//     RulliCentroTagliTask Inputs/RULLI_CENTRO_TAGLI.Catenaria_C4_Rotazione_Status_Dword/InTargetPosition <-> Outputs/ToPlc/StateDWord/InTargetPosition
//     RulliCentroTagliTask Inputs/RULLI_CENTRO_TAGLI.Catenaria_C4_Rotazione_Status_Dword/IoDataInvalid <-> Outputs/ToPlc/StateDWord/IoDataInvalid
//     RulliCentroTagliTask Inputs/RULLI_CENTRO_TAGLI.Catenaria_C4_Rotazione_Status_Dword/MotionCommandsLocked <-> Outputs/ToPlc/StateDWord/MotionCommandsLocked
//     RulliCentroTagliTask Inputs/RULLI_CENTRO_TAGLI.Catenaria_C4_Rotazione_Status_Dword/NegativeDirection <-> Outputs/ToPlc/StateDWord/NegativeDirection
//     RulliCentroTagliTask Inputs/RULLI_CENTRO_TAGLI.Catenaria_C4_Rotazione_Status_Dword/NewTargetPos <-> Outputs/ToPlc/StateDWord/NewTargetPos
//     RulliCentroTagliTask Inputs/RULLI_CENTRO_TAGLI.Catenaria_C4_Rotazione_Status_Dword/NotMoving <-> Outputs/ToPlc/StateDWord/NotMoving
//     RulliCentroTagliTask Inputs/RULLI_CENTRO_TAGLI.Catenaria_C4_Rotazione_Status_Dword/Operational <-> Outputs/ToPlc/StateDWord/Operational
//     RulliCentroTagliTask Inputs/RULLI_CENTRO_TAGLI.Catenaria_C4_Rotazione_Status_Dword/PTPmode <-> Outputs/ToPlc/StateDWord/PTPmode
//     RulliCentroTagliTask Inputs/RULLI_CENTRO_TAGLI.Catenaria_C4_Rotazione_Status_Dword/PhasingActive <-> Outputs/ToPlc/StateDWord/PhasingActive
//     RulliCentroTagliTask Inputs/RULLI_CENTRO_TAGLI.Catenaria_C4_Rotazione_Status_Dword/PositiveDirection <-> Outputs/ToPlc/StateDWord/PositiveDirection
//     RulliCentroTagliTask Inputs/RULLI_CENTRO_TAGLI.Catenaria_C4_Rotazione_Status_Dword/Protected_ <-> Outputs/ToPlc/StateDWord/Protected
//     RulliCentroTagliTask Inputs/RULLI_CENTRO_TAGLI.Catenaria_C4_Rotazione_Status_Dword/SoftLimitMaxExceeded <-> Outputs/ToPlc/StateDWord/SoftLimitMaxExceeded
//     RulliCentroTagliTask Inputs/RULLI_CENTRO_TAGLI.Catenaria_C4_Rotazione_Status_Dword/SoftLimitMinExceeded <-> Outputs/ToPlc/StateDWord/SoftLimitMinExceeded
//     RulliCentroTagliTask Outputs/RULLI_CENTRO_TAGLI.Catenaria_C4_Rotazione.PlcToNc <-> Inputs/FromPlc
//   Galimberti/Galimberti Instance <-> NC-Task 1 SAF/Axes/C5
//     RulliCentroTagliTask Inputs/RULLI_CENTRO_TAGLI.Catenaria_C5_Rotazione.NcToPlc <-> Outputs/ToPlc
//     RulliCentroTagliTask Inputs/RULLI_CENTRO_TAGLI.Catenaria_C5_Rotazione_Status_Dword/CamDataQueued <-> Outputs/ToPlc/StateDWord/CamDataQueued
//     RulliCentroTagliTask Inputs/RULLI_CENTRO_TAGLI.Catenaria_C5_Rotazione_Status_Dword/CamScalingPending <-> Outputs/ToPlc/StateDWord/CamScalingPending
//     RulliCentroTagliTask Inputs/RULLI_CENTRO_TAGLI.Catenaria_C5_Rotazione_Status_Dword/CamTableQueued <-> Outputs/ToPlc/StateDWord/CamTableQueued
//     RulliCentroTagliTask Inputs/RULLI_CENTRO_TAGLI.Catenaria_C5_Rotazione_Status_Dword/CmdBuffered <-> Outputs/ToPlc/StateDWord/CmdBuffered
//     RulliCentroTagliTask Inputs/RULLI_CENTRO_TAGLI.Catenaria_C5_Rotazione_Status_Dword/Compensating <-> Outputs/ToPlc/StateDWord/Compensating
//     RulliCentroTagliTask Inputs/RULLI_CENTRO_TAGLI.Catenaria_C5_Rotazione_Status_Dword/ConstantVelocity <-> Outputs/ToPlc/StateDWord/ConstantVelocity
//     RulliCentroTagliTask Inputs/RULLI_CENTRO_TAGLI.Catenaria_C5_Rotazione_Status_Dword/ContinuousMotion <-> Outputs/ToPlc/StateDWord/ContinuousMotion
//     RulliCentroTagliTask Inputs/RULLI_CENTRO_TAGLI.Catenaria_C5_Rotazione_Status_Dword/ControlLoopClosed <-> Outputs/ToPlc/StateDWord/ControlLoopClosed
//     RulliCentroTagliTask Inputs/RULLI_CENTRO_TAGLI.Catenaria_C5_Rotazione_Status_Dword/DriveDeviceError <-> Outputs/ToPlc/StateDWord/DriveDeviceError
//     RulliCentroTagliTask Inputs/RULLI_CENTRO_TAGLI.Catenaria_C5_Rotazione_Status_Dword/Error <-> Outputs/ToPlc/StateDWord/Error
//     RulliCentroTagliTask Inputs/RULLI_CENTRO_TAGLI.Catenaria_C5_Rotazione_Status_Dword/ErrorPropagationDelayed <-> Outputs/ToPlc/StateDWord/ErrorPropagationDelayed
//     RulliCentroTagliTask Inputs/RULLI_CENTRO_TAGLI.Catenaria_C5_Rotazione_Status_Dword/ExtSetPointGenEnabled <-> Outputs/ToPlc/StateDWord/ExtSetPointGenEnabled
//     RulliCentroTagliTask Inputs/RULLI_CENTRO_TAGLI.Catenaria_C5_Rotazione_Status_Dword/ExternalLatchValid <-> Outputs/ToPlc/StateDWord/ExternalLatchValid
//     RulliCentroTagliTask Inputs/RULLI_CENTRO_TAGLI.Catenaria_C5_Rotazione_Status_Dword/HasBeenStopped <-> Outputs/ToPlc/StateDWord/HasBeenStopped
//     RulliCentroTagliTask Inputs/RULLI_CENTRO_TAGLI.Catenaria_C5_Rotazione_Status_Dword/HasJob <-> Outputs/ToPlc/StateDWord/HasJob
//     RulliCentroTagliTask Inputs/RULLI_CENTRO_TAGLI.Catenaria_C5_Rotazione_Status_Dword/Homed <-> Outputs/ToPlc/StateDWord/Homed
//     RulliCentroTagliTask Inputs/RULLI_CENTRO_TAGLI.Catenaria_C5_Rotazione_Status_Dword/HomingBusy <-> Outputs/ToPlc/StateDWord/HomingBusy
//     RulliCentroTagliTask Inputs/RULLI_CENTRO_TAGLI.Catenaria_C5_Rotazione_Status_Dword/InPositionArea <-> Outputs/ToPlc/StateDWord/InPositionArea
//     RulliCentroTagliTask Inputs/RULLI_CENTRO_TAGLI.Catenaria_C5_Rotazione_Status_Dword/InTargetPosition <-> Outputs/ToPlc/StateDWord/InTargetPosition
//     RulliCentroTagliTask Inputs/RULLI_CENTRO_TAGLI.Catenaria_C5_Rotazione_Status_Dword/IoDataInvalid <-> Outputs/ToPlc/StateDWord/IoDataInvalid
//     RulliCentroTagliTask Inputs/RULLI_CENTRO_TAGLI.Catenaria_C5_Rotazione_Status_Dword/MotionCommandsLocked <-> Outputs/ToPlc/StateDWord/MotionCommandsLocked
//     RulliCentroTagliTask Inputs/RULLI_CENTRO_TAGLI.Catenaria_C5_Rotazione_Status_Dword/NegativeDirection <-> Outputs/ToPlc/StateDWord/NegativeDirection
//     RulliCentroTagliTask Inputs/RULLI_CENTRO_TAGLI.Catenaria_C5_Rotazione_Status_Dword/NewTargetPos <-> Outputs/ToPlc/StateDWord/NewTargetPos
//     RulliCentroTagliTask Inputs/RULLI_CENTRO_TAGLI.Catenaria_C5_Rotazione_Status_Dword/NotMoving <-> Outputs/ToPlc/StateDWord/NotMoving
//     RulliCentroTagliTask Inputs/RULLI_CENTRO_TAGLI.Catenaria_C5_Rotazione_Status_Dword/Operational <-> Outputs/ToPlc/StateDWord/Operational
//     RulliCentroTagliTask Inputs/RULLI_CENTRO_TAGLI.Catenaria_C5_Rotazione_Status_Dword/PTPmode <-> Outputs/ToPlc/StateDWord/PTPmode
//     RulliCentroTagliTask Inputs/RULLI_CENTRO_TAGLI.Catenaria_C5_Rotazione_Status_Dword/PhasingActive <-> Outputs/ToPlc/StateDWord/PhasingActive
//     RulliCentroTagliTask Inputs/RULLI_CENTRO_TAGLI.Catenaria_C5_Rotazione_Status_Dword/PositiveDirection <-> Outputs/ToPlc/StateDWord/PositiveDirection
//     RulliCentroTagliTask Inputs/RULLI_CENTRO_TAGLI.Catenaria_C5_Rotazione_Status_Dword/Protected_ <-> Outputs/ToPlc/StateDWord/Protected
//     RulliCentroTagliTask Inputs/RULLI_CENTRO_TAGLI.Catenaria_C5_Rotazione_Status_Dword/SoftLimitMaxExceeded <-> Outputs/ToPlc/StateDWord/SoftLimitMaxExceeded
//     RulliCentroTagliTask Inputs/RULLI_CENTRO_TAGLI.Catenaria_C5_Rotazione_Status_Dword/SoftLimitMinExceeded <-> Outputs/ToPlc/StateDWord/SoftLimitMinExceeded
//     RulliCentroTagliTask Outputs/RULLI_CENTRO_TAGLI.Catenaria_C5_Rotazione.PlcToNc <-> Inputs/FromPlc
//   Galimberti/Galimberti Instance <-> NC-Task 1 SAF/Axes/C6
//     RulliCentroTagliTask Inputs/RULLI_CENTRO_TAGLI.Catenaria_C6_Rotazione.NcToPlc <-> Outputs/ToPlc
//     RulliCentroTagliTask Inputs/RULLI_CENTRO_TAGLI.Catenaria_C6_Rotazione_Status_Dword/CamDataQueued <-> Outputs/ToPlc/StateDWord/CamDataQueued
//     RulliCentroTagliTask Inputs/RULLI_CENTRO_TAGLI.Catenaria_C6_Rotazione_Status_Dword/CamScalingPending <-> Outputs/ToPlc/StateDWord/CamScalingPending
//     RulliCentroTagliTask Inputs/RULLI_CENTRO_TAGLI.Catenaria_C6_Rotazione_Status_Dword/CamTableQueued <-> Outputs/ToPlc/StateDWord/CamTableQueued
//     RulliCentroTagliTask Inputs/RULLI_CENTRO_TAGLI.Catenaria_C6_Rotazione_Status_Dword/CmdBuffered <-> Outputs/ToPlc/StateDWord/CmdBuffered
//     RulliCentroTagliTask Inputs/RULLI_CENTRO_TAGLI.Catenaria_C6_Rotazione_Status_Dword/Compensating <-> Outputs/ToPlc/StateDWord/Compensating
//     RulliCentroTagliTask Inputs/RULLI_CENTRO_TAGLI.Catenaria_C6_Rotazione_Status_Dword/ConstantVelocity <-> Outputs/ToPlc/StateDWord/ConstantVelocity
//     RulliCentroTagliTask Inputs/RULLI_CENTRO_TAGLI.Catenaria_C6_Rotazione_Status_Dword/ContinuousMotion <-> Outputs/ToPlc/StateDWord/ContinuousMotion
//     RulliCentroTagliTask Inputs/RULLI_CENTRO_TAGLI.Catenaria_C6_Rotazione_Status_Dword/ControlLoopClosed <-> Outputs/ToPlc/StateDWord/ControlLoopClosed
//     RulliCentroTagliTask Inputs/RULLI_CENTRO_TAGLI.Catenaria_C6_Rotazione_Status_Dword/DriveDeviceError <-> Outputs/ToPlc/StateDWord/DriveDeviceError
//     RulliCentroTagliTask Inputs/RULLI_CENTRO_TAGLI.Catenaria_C6_Rotazione_Status_Dword/Error <-> Outputs/ToPlc/StateDWord/Error
//     RulliCentroTagliTask Inputs/RULLI_CENTRO_TAGLI.Catenaria_C6_Rotazione_Status_Dword/ErrorPropagationDelayed <-> Outputs/ToPlc/StateDWord/ErrorPropagationDelayed
//     RulliCentroTagliTask Inputs/RULLI_CENTRO_TAGLI.Catenaria_C6_Rotazione_Status_Dword/ExtSetPointGenEnabled <-> Outputs/ToPlc/StateDWord/ExtSetPointGenEnabled
//     RulliCentroTagliTask Inputs/RULLI_CENTRO_TAGLI.Catenaria_C6_Rotazione_Status_Dword/ExternalLatchValid <-> Outputs/ToPlc/StateDWord/ExternalLatchValid
//     RulliCentroTagliTask Inputs/RULLI_CENTRO_TAGLI.Catenaria_C6_Rotazione_Status_Dword/HasBeenStopped <-> Outputs/ToPlc/StateDWord/HasBeenStopped
//     RulliCentroTagliTask Inputs/RULLI_CENTRO_TAGLI.Catenaria_C6_Rotazione_Status_Dword/HasJob <-> Outputs/ToPlc/StateDWord/HasJob
//     RulliCentroTagliTask Inputs/RULLI_CENTRO_TAGLI.Catenaria_C6_Rotazione_Status_Dword/Homed <-> Outputs/ToPlc/StateDWord/Homed
//     RulliCentroTagliTask Inputs/RULLI_CENTRO_TAGLI.Catenaria_C6_Rotazione_Status_Dword/HomingBusy <-> Outputs/ToPlc/StateDWord/HomingBusy
//     RulliCentroTagliTask Inputs/RULLI_CENTRO_TAGLI.Catenaria_C6_Rotazione_Status_Dword/InPositionArea <-> Outputs/ToPlc/StateDWord/InPositionArea
//     RulliCentroTagliTask Inputs/RULLI_CENTRO_TAGLI.Catenaria_C6_Rotazione_Status_Dword/InTargetPosition <-> Outputs/ToPlc/StateDWord/InTargetPosition
//     RulliCentroTagliTask Inputs/RULLI_CENTRO_TAGLI.Catenaria_C6_Rotazione_Status_Dword/IoDataInvalid <-> Outputs/ToPlc/StateDWord/IoDataInvalid
//     RulliCentroTagliTask Inputs/RULLI_CENTRO_TAGLI.Catenaria_C6_Rotazione_Status_Dword/MotionCommandsLocked <-> Outputs/ToPlc/StateDWord/MotionCommandsLocked
//     RulliCentroTagliTask Inputs/RULLI_CENTRO_TAGLI.Catenaria_C6_Rotazione_Status_Dword/NegativeDirection <-> Outputs/ToPlc/StateDWord/NegativeDirection
//     RulliCentroTagliTask Inputs/RULLI_CENTRO_TAGLI.Catenaria_C6_Rotazione_Status_Dword/NewTargetPos <-> Outputs/ToPlc/StateDWord/NewTargetPos
//     RulliCentroTagliTask Inputs/RULLI_CENTRO_TAGLI.Catenaria_C6_Rotazione_Status_Dword/NotMoving <-> Outputs/ToPlc/StateDWord/NotMoving
//     RulliCentroTagliTask Inputs/RULLI_CENTRO_TAGLI.Catenaria_C6_Rotazione_Status_Dword/Operational <-> Outputs/ToPlc/StateDWord/Operational
//     RulliCentroTagliTask Inputs/RULLI_CENTRO_TAGLI.Catenaria_C6_Rotazione_Status_Dword/PTPmode <-> Outputs/ToPlc/StateDWord/PTPmode
//     RulliCentroTagliTask Inputs/RULLI_CENTRO_TAGLI.Catenaria_C6_Rotazione_Status_Dword/PhasingActive <-> Outputs/ToPlc/StateDWord/PhasingActive
//     RulliCentroTagliTask Inputs/RULLI_CENTRO_TAGLI.Catenaria_C6_Rotazione_Status_Dword/PositiveDirection <-> Outputs/ToPlc/StateDWord/PositiveDirection
//     RulliCentroTagliTask Inputs/RULLI_CENTRO_TAGLI.Catenaria_C6_Rotazione_Status_Dword/Protected_ <-> Outputs/ToPlc/StateDWord/Protected
//     RulliCentroTagliTask Inputs/RULLI_CENTRO_TAGLI.Catenaria_C6_Rotazione_Status_Dword/SoftLimitMaxExceeded <-> Outputs/ToPlc/StateDWord/SoftLimitMaxExceeded
//     RulliCentroTagliTask Inputs/RULLI_CENTRO_TAGLI.Catenaria_C6_Rotazione_Status_Dword/SoftLimitMinExceeded <-> Outputs/ToPlc/StateDWord/SoftLimitMinExceeded
//     RulliCentroTagliTask Outputs/RULLI_CENTRO_TAGLI.Catenaria_C6_Rotazione.PlcToNc <-> Inputs/FromPlc
//   Galimberti/Galimberti Instance <-> NC-Task 1 SAF/Axes/R1M1
//     RulliCentroTagliTask Inputs/RULLI_CENTRO_TAGLI.Rulliera_R1_Rotazione.NcToPlc <-> Outputs/ToPlc
//     RulliCentroTagliTask Inputs/RULLI_CENTRO_TAGLI.Rulliera_R1_Rotazione_Status_Dword/CamDataQueued <-> Outputs/ToPlc/StateDWord/CamDataQueued
//     RulliCentroTagliTask Inputs/RULLI_CENTRO_TAGLI.Rulliera_R1_Rotazione_Status_Dword/CamScalingPending <-> Outputs/ToPlc/StateDWord/CamScalingPending
//     RulliCentroTagliTask Inputs/RULLI_CENTRO_TAGLI.Rulliera_R1_Rotazione_Status_Dword/CamTableQueued <-> Outputs/ToPlc/StateDWord/CamTableQueued
//     RulliCentroTagliTask Inputs/RULLI_CENTRO_TAGLI.Rulliera_R1_Rotazione_Status_Dword/CmdBuffered <-> Outputs/ToPlc/StateDWord/CmdBuffered
//     RulliCentroTagliTask Inputs/RULLI_CENTRO_TAGLI.Rulliera_R1_Rotazione_Status_Dword/Compensating <-> Outputs/ToPlc/StateDWord/Compensating
//     RulliCentroTagliTask Inputs/RULLI_CENTRO_TAGLI.Rulliera_R1_Rotazione_Status_Dword/ConstantVelocity <-> Outputs/ToPlc/StateDWord/ConstantVelocity
//     RulliCentroTagliTask Inputs/RULLI_CENTRO_TAGLI.Rulliera_R1_Rotazione_Status_Dword/ContinuousMotion <-> Outputs/ToPlc/StateDWord/ContinuousMotion
//     RulliCentroTagliTask Inputs/RULLI_CENTRO_TAGLI.Rulliera_R1_Rotazione_Status_Dword/ControlLoopClosed <-> Outputs/ToPlc/StateDWord/ControlLoopClosed
//     RulliCentroTagliTask Inputs/RULLI_CENTRO_TAGLI.Rulliera_R1_Rotazione_Status_Dword/DriveDeviceError <-> Outputs/ToPlc/StateDWord/DriveDeviceError
//     RulliCentroTagliTask Inputs/RULLI_CENTRO_TAGLI.Rulliera_R1_Rotazione_Status_Dword/Error <-> Outputs/ToPlc/StateDWord/Error
//     RulliCentroTagliTask Inputs/RULLI_CENTRO_TAGLI.Rulliera_R1_Rotazione_Status_Dword/ErrorPropagationDelayed <-> Outputs/ToPlc/StateDWord/ErrorPropagationDelayed
//     RulliCentroTagliTask Inputs/RULLI_CENTRO_TAGLI.Rulliera_R1_Rotazione_Status_Dword/ExtSetPointGenEnabled <-> Outputs/ToPlc/StateDWord/ExtSetPointGenEnabled
//     RulliCentroTagliTask Inputs/RULLI_CENTRO_TAGLI.Rulliera_R1_Rotazione_Status_Dword/ExternalLatchValid <-> Outputs/ToPlc/StateDWord/ExternalLatchValid
//     RulliCentroTagliTask Inputs/RULLI_CENTRO_TAGLI.Rulliera_R1_Rotazione_Status_Dword/HasBeenStopped <-> Outputs/ToPlc/StateDWord/HasBeenStopped
//     RulliCentroTagliTask Inputs/RULLI_CENTRO_TAGLI.Rulliera_R1_Rotazione_Status_Dword/HasJob <-> Outputs/ToPlc/StateDWord/HasJob
//     RulliCentroTagliTask Inputs/RULLI_CENTRO_TAGLI.Rulliera_R1_Rotazione_Status_Dword/Homed <-> Outputs/ToPlc/StateDWord/Homed
//     RulliCentroTagliTask Inputs/RULLI_CENTRO_TAGLI.Rulliera_R1_Rotazione_Status_Dword/HomingBusy <-> Outputs/ToPlc/StateDWord/HomingBusy
//     RulliCentroTagliTask Inputs/RULLI_CENTRO_TAGLI.Rulliera_R1_Rotazione_Status_Dword/InPositionArea <-> Outputs/ToPlc/StateDWord/InPositionArea
//     RulliCentroTagliTask Inputs/RULLI_CENTRO_TAGLI.Rulliera_R1_Rotazione_Status_Dword/InTargetPosition <-> Outputs/ToPlc/StateDWord/InTargetPosition
//     RulliCentroTagliTask Inputs/RULLI_CENTRO_TAGLI.Rulliera_R1_Rotazione_Status_Dword/IoDataInvalid <-> Outputs/ToPlc/StateDWord/IoDataInvalid
//     RulliCentroTagliTask Inputs/RULLI_CENTRO_TAGLI.Rulliera_R1_Rotazione_Status_Dword/MotionCommandsLocked <-> Outputs/ToPlc/StateDWord/MotionCommandsLocked
//     RulliCentroTagliTask Inputs/RULLI_CENTRO_TAGLI.Rulliera_R1_Rotazione_Status_Dword/NegativeDirection <-> Outputs/ToPlc/StateDWord/NegativeDirection
//     RulliCentroTagliTask Inputs/RULLI_CENTRO_TAGLI.Rulliera_R1_Rotazione_Status_Dword/NewTargetPos <-> Outputs/ToPlc/StateDWord/NewTargetPos
//     RulliCentroTagliTask Inputs/RULLI_CENTRO_TAGLI.Rulliera_R1_Rotazione_Status_Dword/NotMoving <-> Outputs/ToPlc/StateDWord/NotMoving
//     RulliCentroTagliTask Inputs/RULLI_CENTRO_TAGLI.Rulliera_R1_Rotazione_Status_Dword/Operational <-> Outputs/ToPlc/StateDWord/Operational
//     RulliCentroTagliTask Inputs/RULLI_CENTRO_TAGLI.Rulliera_R1_Rotazione_Status_Dword/PTPmode <-> Outputs/ToPlc/StateDWord/PTPmode
//     RulliCentroTagliTask Inputs/RULLI_CENTRO_TAGLI.Rulliera_R1_Rotazione_Status_Dword/PhasingActive <-> Outputs/ToPlc/StateDWord/PhasingActive
//     RulliCentroTagliTask Inputs/RULLI_CENTRO_TAGLI.Rulliera_R1_Rotazione_Status_Dword/PositiveDirection <-> Outputs/ToPlc/StateDWord/PositiveDirection
//     RulliCentroTagliTask Inputs/RULLI_CENTRO_TAGLI.Rulliera_R1_Rotazione_Status_Dword/Protected_ <-> Outputs/ToPlc/StateDWord/Protected
//     RulliCentroTagliTask Inputs/RULLI_CENTRO_TAGLI.Rulliera_R1_Rotazione_Status_Dword/SoftLimitMaxExceeded <-> Outputs/ToPlc/StateDWord/SoftLimitMaxExceeded
//     RulliCentroTagliTask Inputs/RULLI_CENTRO_TAGLI.Rulliera_R1_Rotazione_Status_Dword/SoftLimitMinExceeded <-> Outputs/ToPlc/StateDWord/SoftLimitMinExceeded
//     RulliCentroTagliTask Outputs/RULLI_CENTRO_TAGLI.Rulliera_R1_Rotazione.PlcToNc <-> Inputs/FromPlc
//   Galimberti/Galimberti Instance <-> NC-Task 1 SAF/Axes/R2
//     RulliCentroTagliTask Inputs/RULLI_CENTRO_TAGLI.Rulliera_R2_Act_Pos <-> Outputs/ToPlc/ActPos
//     RulliCentroTagliTask Inputs/RULLI_CENTRO_TAGLI.Rulliera_R2_Rotazione.NcToPlc <-> Outputs/ToPlc
//     RulliCentroTagliTask Inputs/RULLI_CENTRO_TAGLI.Rulliera_R2_Rotazione_Status_Dword/CamDataQueued <-> Outputs/ToPlc/StateDWord/CamDataQueued
//     RulliCentroTagliTask Inputs/RULLI_CENTRO_TAGLI.Rulliera_R2_Rotazione_Status_Dword/CamScalingPending <-> Outputs/ToPlc/StateDWord/CamScalingPending
//     RulliCentroTagliTask Inputs/RULLI_CENTRO_TAGLI.Rulliera_R2_Rotazione_Status_Dword/CamTableQueued <-> Outputs/ToPlc/StateDWord/CamTableQueued
//     RulliCentroTagliTask Inputs/RULLI_CENTRO_TAGLI.Rulliera_R2_Rotazione_Status_Dword/CmdBuffered <-> Outputs/ToPlc/StateDWord/CmdBuffered
//     RulliCentroTagliTask Inputs/RULLI_CENTRO_TAGLI.Rulliera_R2_Rotazione_Status_Dword/Compensating <-> Outputs/ToPlc/StateDWord/Compensating
//     RulliCentroTagliTask Inputs/RULLI_CENTRO_TAGLI.Rulliera_R2_Rotazione_Status_Dword/ConstantVelocity <-> Outputs/ToPlc/StateDWord/ConstantVelocity
//     RulliCentroTagliTask Inputs/RULLI_CENTRO_TAGLI.Rulliera_R2_Rotazione_Status_Dword/ContinuousMotion <-> Outputs/ToPlc/StateDWord/ContinuousMotion
//     RulliCentroTagliTask Inputs/RULLI_CENTRO_TAGLI.Rulliera_R2_Rotazione_Status_Dword/ControlLoopClosed <-> Outputs/ToPlc/StateDWord/ControlLoopClosed
//     RulliCentroTagliTask Inputs/RULLI_CENTRO_TAGLI.Rulliera_R2_Rotazione_Status_Dword/DriveDeviceError <-> Outputs/ToPlc/StateDWord/DriveDeviceError
//     RulliCentroTagliTask Inputs/RULLI_CENTRO_TAGLI.Rulliera_R2_Rotazione_Status_Dword/Error <-> Outputs/ToPlc/StateDWord/Error
//     RulliCentroTagliTask Inputs/RULLI_CENTRO_TAGLI.Rulliera_R2_Rotazione_Status_Dword/ErrorPropagationDelayed <-> Outputs/ToPlc/StateDWord/ErrorPropagationDelayed
//     RulliCentroTagliTask Inputs/RULLI_CENTRO_TAGLI.Rulliera_R2_Rotazione_Status_Dword/ExtSetPointGenEnabled <-> Outputs/ToPlc/StateDWord/ExtSetPointGenEnabled
//     RulliCentroTagliTask Inputs/RULLI_CENTRO_TAGLI.Rulliera_R2_Rotazione_Status_Dword/ExternalLatchValid <-> Outputs/ToPlc/StateDWord/ExternalLatchValid
//     RulliCentroTagliTask Inputs/RULLI_CENTRO_TAGLI.Rulliera_R2_Rotazione_Status_Dword/HasBeenStopped <-> Outputs/ToPlc/StateDWord/HasBeenStopped
//     RulliCentroTagliTask Inputs/RULLI_CENTRO_TAGLI.Rulliera_R2_Rotazione_Status_Dword/HasJob <-> Outputs/ToPlc/StateDWord/HasJob
//     RulliCentroTagliTask Inputs/RULLI_CENTRO_TAGLI.Rulliera_R2_Rotazione_Status_Dword/Homed <-> Outputs/ToPlc/StateDWord/Homed
//     RulliCentroTagliTask Inputs/RULLI_CENTRO_TAGLI.Rulliera_R2_Rotazione_Status_Dword/HomingBusy <-> Outputs/ToPlc/StateDWord/HomingBusy
//     RulliCentroTagliTask Inputs/RULLI_CENTRO_TAGLI.Rulliera_R2_Rotazione_Status_Dword/InPositionArea <-> Outputs/ToPlc/StateDWord/InPositionArea
//     RulliCentroTagliTask Inputs/RULLI_CENTRO_TAGLI.Rulliera_R2_Rotazione_Status_Dword/InTargetPosition <-> Outputs/ToPlc/StateDWord/InTargetPosition
//     RulliCentroTagliTask Inputs/RULLI_CENTRO_TAGLI.Rulliera_R2_Rotazione_Status_Dword/IoDataInvalid <-> Outputs/ToPlc/StateDWord/IoDataInvalid
//     RulliCentroTagliTask Inputs/RULLI_CENTRO_TAGLI.Rulliera_R2_Rotazione_Status_Dword/MotionCommandsLocked <-> Outputs/ToPlc/StateDWord/MotionCommandsLocked
//     RulliCentroTagliTask Inputs/RULLI_CENTRO_TAGLI.Rulliera_R2_Rotazione_Status_Dword/NegativeDirection <-> Outputs/ToPlc/StateDWord/NegativeDirection
//     RulliCentroTagliTask Inputs/RULLI_CENTRO_TAGLI.Rulliera_R2_Rotazione_Status_Dword/NewTargetPos <-> Outputs/ToPlc/StateDWord/NewTargetPos
//     RulliCentroTagliTask Inputs/RULLI_CENTRO_TAGLI.Rulliera_R2_Rotazione_Status_Dword/NotMoving <-> Outputs/ToPlc/StateDWord/NotMoving
//     RulliCentroTagliTask Inputs/RULLI_CENTRO_TAGLI.Rulliera_R2_Rotazione_Status_Dword/Operational <-> Outputs/ToPlc/StateDWord/Operational
//     RulliCentroTagliTask Inputs/RULLI_CENTRO_TAGLI.Rulliera_R2_Rotazione_Status_Dword/PTPmode <-> Outputs/ToPlc/StateDWord/PTPmode
//     RulliCentroTagliTask Inputs/RULLI_CENTRO_TAGLI.Rulliera_R2_Rotazione_Status_Dword/PhasingActive <-> Outputs/ToPlc/StateDWord/PhasingActive
//     RulliCentroTagliTask Inputs/RULLI_CENTRO_TAGLI.Rulliera_R2_Rotazione_Status_Dword/PositiveDirection <-> Outputs/ToPlc/StateDWord/PositiveDirection
//     RulliCentroTagliTask Inputs/RULLI_CENTRO_TAGLI.Rulliera_R2_Rotazione_Status_Dword/Protected_ <-> Outputs/ToPlc/StateDWord/Protected
//     RulliCentroTagliTask Inputs/RULLI_CENTRO_TAGLI.Rulliera_R2_Rotazione_Status_Dword/SoftLimitMaxExceeded <-> Outputs/ToPlc/StateDWord/SoftLimitMaxExceeded
//     RulliCentroTagliTask Inputs/RULLI_CENTRO_TAGLI.Rulliera_R2_Rotazione_Status_Dword/SoftLimitMinExceeded <-> Outputs/ToPlc/StateDWord/SoftLimitMinExceeded
//     RulliCentroTagliTask Outputs/RULLI_CENTRO_TAGLI.Rulliera_R2_Rotazione.PlcToNc <-> Inputs/FromPlc
//   Galimberti/Galimberti Instance <-> NC-Task 1 SAF/Axes/R3
//     RulliCentroTagliTask Inputs/RULLI_CENTRO_TAGLI.Rulliera_R3_Rotazione.NcToPlc <-> Outputs/ToPlc
//     RulliCentroTagliTask Inputs/RULLI_CENTRO_TAGLI.Rulliera_R3_Rotazione_Status_Dword/CamDataQueued <-> Outputs/ToPlc/StateDWord/CamDataQueued
//     RulliCentroTagliTask Inputs/RULLI_CENTRO_TAGLI.Rulliera_R3_Rotazione_Status_Dword/CamScalingPending <-> Outputs/ToPlc/StateDWord/CamScalingPending
//     RulliCentroTagliTask Inputs/RULLI_CENTRO_TAGLI.Rulliera_R3_Rotazione_Status_Dword/CamTableQueued <-> Outputs/ToPlc/StateDWord/CamTableQueued
//     RulliCentroTagliTask Inputs/RULLI_CENTRO_TAGLI.Rulliera_R3_Rotazione_Status_Dword/CmdBuffered <-> Outputs/ToPlc/StateDWord/CmdBuffered
//     RulliCentroTagliTask Inputs/RULLI_CENTRO_TAGLI.Rulliera_R3_Rotazione_Status_Dword/Compensating <-> Outputs/ToPlc/StateDWord/Compensating
//     RulliCentroTagliTask Inputs/RULLI_CENTRO_TAGLI.Rulliera_R3_Rotazione_Status_Dword/ConstantVelocity <-> Outputs/ToPlc/StateDWord/ConstantVelocity
//     RulliCentroTagliTask Inputs/RULLI_CENTRO_TAGLI.Rulliera_R3_Rotazione_Status_Dword/ContinuousMotion <-> Outputs/ToPlc/StateDWord/ContinuousMotion
//     RulliCentroTagliTask Inputs/RULLI_CENTRO_TAGLI.Rulliera_R3_Rotazione_Status_Dword/ControlLoopClosed <-> Outputs/ToPlc/StateDWord/ControlLoopClosed
//     RulliCentroTagliTask Inputs/RULLI_CENTRO_TAGLI.Rulliera_R3_Rotazione_Status_Dword/DriveDeviceError <-> Outputs/ToPlc/StateDWord/DriveDeviceError
//     RulliCentroTagliTask Inputs/RULLI_CENTRO_TAGLI.Rulliera_R3_Rotazione_Status_Dword/Error <-> Outputs/ToPlc/StateDWord/Error
//     RulliCentroTagliTask Inputs/RULLI_CENTRO_TAGLI.Rulliera_R3_Rotazione_Status_Dword/ErrorPropagationDelayed <-> Outputs/ToPlc/StateDWord/ErrorPropagationDelayed
//     RulliCentroTagliTask Inputs/RULLI_CENTRO_TAGLI.Rulliera_R3_Rotazione_Status_Dword/ExtSetPointGenEnabled <-> Outputs/ToPlc/StateDWord/ExtSetPointGenEnabled
//     RulliCentroTagliTask Inputs/RULLI_CENTRO_TAGLI.Rulliera_R3_Rotazione_Status_Dword/ExternalLatchValid <-> Outputs/ToPlc/StateDWord/ExternalLatchValid
//     RulliCentroTagliTask Inputs/RULLI_CENTRO_TAGLI.Rulliera_R3_Rotazione_Status_Dword/HasBeenStopped <-> Outputs/ToPlc/StateDWord/HasBeenStopped
//     RulliCentroTagliTask Inputs/RULLI_CENTRO_TAGLI.Rulliera_R3_Rotazione_Status_Dword/HasJob <-> Outputs/ToPlc/StateDWord/HasJob
//     RulliCentroTagliTask Inputs/RULLI_CENTRO_TAGLI.Rulliera_R3_Rotazione_Status_Dword/Homed <-> Outputs/ToPlc/StateDWord/Homed
//     RulliCentroTagliTask Inputs/RULLI_CENTRO_TAGLI.Rulliera_R3_Rotazione_Status_Dword/HomingBusy <-> Outputs/ToPlc/StateDWord/HomingBusy
//     RulliCentroTagliTask Inputs/RULLI_CENTRO_TAGLI.Rulliera_R3_Rotazione_Status_Dword/InPositionArea <-> Outputs/ToPlc/StateDWord/InPositionArea
//     RulliCentroTagliTask Inputs/RULLI_CENTRO_TAGLI.Rulliera_R3_Rotazione_Status_Dword/InTargetPosition <-> Outputs/ToPlc/StateDWord/InTargetPosition
//     RulliCentroTagliTask Inputs/RULLI_CENTRO_TAGLI.Rulliera_R3_Rotazione_Status_Dword/IoDataInvalid <-> Outputs/ToPlc/StateDWord/IoDataInvalid
//     RulliCentroTagliTask Inputs/RULLI_CENTRO_TAGLI.Rulliera_R3_Rotazione_Status_Dword/MotionCommandsLocked <-> Outputs/ToPlc/StateDWord/MotionCommandsLocked
//     RulliCentroTagliTask Inputs/RULLI_CENTRO_TAGLI.Rulliera_R3_Rotazione_Status_Dword/NegativeDirection <-> Outputs/ToPlc/StateDWord/NegativeDirection
//     RulliCentroTagliTask Inputs/RULLI_CENTRO_TAGLI.Rulliera_R3_Rotazione_Status_Dword/NewTargetPos <-> Outputs/ToPlc/StateDWord/NewTargetPos
//     RulliCentroTagliTask Inputs/RULLI_CENTRO_TAGLI.Rulliera_R3_Rotazione_Status_Dword/NotMoving <-> Outputs/ToPlc/StateDWord/NotMoving
//     RulliCentroTagliTask Inputs/RULLI_CENTRO_TAGLI.Rulliera_R3_Rotazione_Status_Dword/Operational <-> Outputs/ToPlc/StateDWord/Operational
//     RulliCentroTagliTask Inputs/RULLI_CENTRO_TAGLI.Rulliera_R3_Rotazione_Status_Dword/PTPmode <-> Outputs/ToPlc/StateDWord/PTPmode
//     RulliCentroTagliTask Inputs/RULLI_CENTRO_TAGLI.Rulliera_R3_Rotazione_Status_Dword/PhasingActive <-> Outputs/ToPlc/StateDWord/PhasingActive
//     RulliCentroTagliTask Inputs/RULLI_CENTRO_TAGLI.Rulliera_R3_Rotazione_Status_Dword/PositiveDirection <-> Outputs/ToPlc/StateDWord/PositiveDirection
//     RulliCentroTagliTask Inputs/RULLI_CENTRO_TAGLI.Rulliera_R3_Rotazione_Status_Dword/Protected_ <-> Outputs/ToPlc/StateDWord/Protected
//     RulliCentroTagliTask Inputs/RULLI_CENTRO_TAGLI.Rulliera_R3_Rotazione_Status_Dword/SoftLimitMaxExceeded <-> Outputs/ToPlc/StateDWord/SoftLimitMaxExceeded
//     RulliCentroTagliTask Inputs/RULLI_CENTRO_TAGLI.Rulliera_R3_Rotazione_Status_Dword/SoftLimitMinExceeded <-> Outputs/ToPlc/StateDWord/SoftLimitMinExceeded
//     RulliCentroTagliTask Outputs/RULLI_CENTRO_TAGLI.Rulliera_R3_Rotazione.PlcToNc <-> Inputs/FromPlc

CONFIGURATION Galimberti
    RESOURCE PLC ON TwinCAT3
        TASK PlcTask(INTERVAL := T#10ms, PRIORITY := 20);
        TASK RulliCentroTagliTask(INTERVAL := T#10ms, PRIORITY := 21);
        PROGRAM MAIN WITH PlcTask : MAIN;
        PROGRAM MAIN_RCT WITH RulliCentroTagliTask : MAIN_RCT;
    END_RESOURCE
END_CONFIGURATION

// ---- DUTs/EVACUAZIONE SCARTI/ES_ACTVAL.TcDUT
TYPE ES_ACTVAL :
	STRUCT	
		
		//SENSORI
		T3_S1			:INT;	
		T3_S2		 	:INT;	
		S2_S1		 	:INT;
		S1_S02			:INT;	
		T1_S01			:BOOL;

		//STATI		
		PuliziaT1T2_ON			:BOOL;		//STO PULENDO T1 T2 SERVE PER FAR PARTIRE T3
			
	END_STRUCT
END_TYPE

// ---- DUTs/EVACUAZIONE SCARTI/ES_MPO1.TcDUT
TYPE ES_MPO1 :
	STRUCT
		key						:BOOL;	//CHIAVE INSERITA E SU ON
		btn_M_MacOn				:BOOL;	//AVVIO MANUALE MACINATORE
		btn_R_Riarmo			:BOOL;	//area m armata e ready
		btn_0_AreaMoff			:BOOL;	//SPEGNIMENTO UTENZE PULSANTIERA MP01
		btn_Fsx_T3StartMan		:BOOL;	//AVVIO T3 MANUALE
		btn_Fsx_T4StartMan		:BOOL;	//AVVIO T4 MANUALE
		btn_Fup_T7Avanti		:BOOL;	//AVVIO T7 MANUALE SALITA
		btn_Fdw_T7Indietro		:BOOL;	//AVVIO T7 MANUALE DISCESA
		led_M_MacOn				:BOOL;	//led pulsante AVVIO MANUALE MACINATORE
		led_R_Riarmo			:BOOL;	//led pulsante area m armata e ready
		led_0_AreaMoff			:BOOL;	//led pulsante SPEGNIMENTO UTENZE PULSANTIERA MP01
	END_STRUCT
END_TYPE

// ---- DUTs/EVACUAZIONE SCARTI/ES_PERSISTENT.TcDUT
TYPE ES_PERSISTENT :
	STRUCT
		
		T1_SO1_distanzaAVuoto	:INT:= 6150;
		T1_SO1_valSoglia		:INT:= 1000;
 
		T3_S1_maxScaleBit		:INT:= 32767; 
		T3_S1_maxScaleIng		:INT:= 1300; 
		T3_S1_deltaLowLimit		:INT:= 30;
		T3_S1_distanzaAVuoto	:INT:= 1230;
		T3_S1_valSoglia			:INT:= 200; 

		T3_S2_maxScaleBit       :INT:= 32767; 
		T3_S2_maxScaleIng		:INT:= 1300; 
		T3_S2_deltaLowLimit		:INT:= 30;
		T3_S2_distanzaAVuoto	:INT:= 590;
		T3_S2_valSoglia			:INT:= 200; 
	
		S2_S1_maxScaleBit       :INT:= 32767; 
		S2_S1_maxScaleIng		:INT:= 6000; 
		S2_S1_deltaLowLimit		:INT:= 30; 
		S2_S1_distanzaAVuoto	:INT:= 6000;
		S2_S1_valSoglia			:INT:= 2000; 

		S1_SO2_maxScaleBit      :INT:= 32767; 
		S1_SO2_maxScaleIng		:INT:= 6000; 
		S1_SO2_deltaLowLimit	:INT:= 30; 
		S1_SO2_distanzaAVuoto	:INT:= 6150;
		S1_SO2_valSoglia		:INT:= 1000; 
		S1_SO2_filtertime		:INT:= 10;	

		T1_Time					:INT:= 5;		//TEMPO SVUOTA T1
		T2_Time					:INT:= 7;		//TEMPO SVUOTA T2
		T3_Time					:INT:= 25;		//TEMPO SVUOTA T3	
	
	END_STRUCT
END_TYPE

// ---- DUTs/EVACUAZIONE SCARTI/ES_M.TcDUT
TYPE ES_M :
STRUCT
END_STRUCT
END_TYPE

// ---- DUTs/EVACUAZIONE SCARTI/ES_ALARM.TcDUT
TYPE ES_ALARM :
	STRUCT
		
		Enable			:BOOL;
		Active			:BOOL;
		Reset			:BOOL;
		tmr				:TON;
		pt				:INT:=7;		//secondi
		
	END_STRUCT
END_TYPE

// ---- DUTs/EVACUAZIONE SCARTI/ES_S1.TcDUT
TYPE ES_S1 :
	STRUCT
		Alarm			:ES_ALARM;		
				
		SO2_actVal		:INT;
		SO2_full		:BOOL;
		SO2_fb			:FB_AnalogSensor_full;	

			
	END_STRUCT
END_TYPE

// ---- DUTs/EVACUAZIONE SCARTI/ES_S1PO1.TcDUT
TYPE ES_S1PO1 :
	STRUCT
		key						:BOOL;	//CHIAVE INSERITA E SU ON
		btn_R_Riarmo			:BOOL;	//area m armata e ready	
		btn_0_AreaMoff			:BOOL;	//SPEGNIMENTO UTENZE PULSANTIERA S1P01
		led_R_Riarmo			:BOOL;	//led pulsante area m armata e ready	
		led_0_AreaMoff			:BOOL;	//led pulsante SPEGNIMENTO UTENZE PULSANTIERA S1P01
	
	END_STRUCT
END_TYPE

// ---- DUTs/EVACUAZIONE SCARTI/ES_S2.TcDUT
TYPE ES_S2 :
	STRUCT
		Alarm			:ES_ALARM;	
			
		S1_actVal		:INT;
		S1_full			:BOOL;
		S1_fb			:FB_AnalogSensor_full;			
	END_STRUCT
END_TYPE

// ---- DUTs/EVACUAZIONE SCARTI/ES_SEMAFORO.TcDUT
TYPE ES_SEMAFORO :
	STRUCT		
		analog0			AT%Q*:USINT;			
		analog1			AT%Q*:USINT;				
		analog2			AT%Q*:USINT;		
		analog3			AT%Q*:USINT;		
		analog4			AT%Q*:USINT;		
		analog5			AT%Q*:USINT;
	END_STRUCT
END_TYPE

// ---- DUTs/EVACUAZIONE SCARTI/ES_T1.TcDUT
TYPE ES_T1 :
	STRUCT
		Alarm			:ES_ALARM;
			
		SO1_actVal		:INT;
		SO1_full		:BOOL;
		SO1_fb			:FB_MMSensor_full;
	END_STRUCT
END_TYPE

// ---- DUTs/EVACUAZIONE SCARTI/ES_T3.TcDUT
TYPE ES_T3 :
	STRUCT
		Alarm			:ES_ALARM;
		
		S1_actVal		:INT;
		S1_full			:BOOL;
		S1_fb			:FB_AnalogSensor_full;	

		S2_actVal		:INT;
		S2_full			:BOOL;
		S2_fb			:FB_AnalogSensor_full;		
	END_STRUCT
END_TYPE

// ---- DUTs/EVACUAZIONE SCARTI/ES_T5.TcDUT
TYPE ES_T5 :
	STRUCT
		Alarm			:ES_ALARM;
	
		S1_rt			:R_TRIG;	
		S1_letto		:BOOL;
	
	END_STRUCT
END_TYPE

// ---- DUTs/EVACUAZIONE SCARTI/ES_T6.TcDUT
TYPE ES_T6 :
	STRUCT
		Alarm			:ES_ALARM;
	
		S1_rt			:R_TRIG;	
		S1_letto		:BOOL;
	END_STRUCT
END_TYPE

// ---- DUTs/RULLI_CENTRO_TAGLI/dut_Axe_Status.TcDUT
TYPE dut_Axe_Status :
STRUCT
	
		Operational				:BOOL;
		Homed					:BOOL;
		NotMoving				:BOOL;
		InPositionArea			:BOOL;
		InTargetPosition		:BOOL;
		Protected_				:BOOL;
		ErrorPropagationDelayed	:BOOL;
		HasBeenStopped			:BOOL;
		HasJob					:BOOL;
		PositiveDirection		:BOOL;
		NegativeDirection		:BOOL;
		HomingBusy				:BOOL;
		ConstantVelocity		:BOOL;
		Compensating			:BOOL;
		ExtSetPointGenEnabled	:BOOL;
		PhasingActive			:BOOL;
		ExternalLatchValid		:BOOL;
		NewTargetPos			:BOOL;
		ContinuousMotion		:BOOL;
		ControlLoopClosed		:BOOL;
		CamTableQueued			:BOOL;
		CamDataQueued			:BOOL;
		CamScalingPending		:BOOL;
		CmdBuffered				:BOOL;
		PTPmode					:BOOL;
		SoftLimitMinExceeded	:BOOL;
		SoftLimitMaxExceeded	:BOOL;
		DriveDeviceError		:BOOL;
		MotionCommandsLocked	:BOOL;
		IoDataInvalid			:BOOL;
		Error					:BOOL;



END_STRUCT
END_TYPE

// ---- DUTs/RULLI_CENTRO_TAGLI/dut_Dati_Pezzo.TcDUT
TYPE dut_Dati_Pezzo :
STRUCT
	
	Busy				:BOOL;
	Rotazione			:INT;   //99=no rotazione - 1=rot. avanti - 2=rot. indietro - 3=doppia rotazione
	Larghezza			:REAL;
	Altezza				:REAL;
	Lunghezza			:REAL;
	Lato_Scarico		:INT;	//1=destra - 2=sinistra
	Nr_Ricetta			:INT;

END_STRUCT
END_TYPE

// ---- GVLs/EVACUAZIONE_SCARTI/GVL_ES_IO.TcGVL
{attribute 'Tc2GvlVarNames'}
VAR_GLOBAL

	glo_ES_VERSION			:STRING:='10.3.0.0';


(*****************************************************************)	
(*****************************************************************)	
(*****************************************************************)	

	//Quadro HQ3
	glo_dig_in_HQ3			AT %I*:ARRAY[1..64] OF BOOL;
	glo_dig_out_HQ3			AT %Q*:ARRAY[1..64] OF BOOL;
	glo_WcState_HQ3			AT %I*:ARRAY[1..64] OF BOOL;	//0:Valid, 1:Invalid
	glo_State_HQ3			AT %I*:ARRAY[1..64] OF UINT;	//8:OP
	
	
(*****************************************************************)	
(*****************************************************************)	
(*****************************************************************)	

	//Quadro HQ1	
	glo_dig_in_HQ1			AT %I*:ARRAY[1..64] OF BOOL;
	glo_dig_out_HQ1			AT %Q*:ARRAY[1..64] OF BOOL;	
	glo_analog_in_HQ1		AT %I*:ARRAY[1..64] OF INT;
	glo_WcState_HQ1			AT %I*:ARRAY[1..64] OF BOOL;	//0:Valid, 1:Invalid
	glo_State_HQ1			AT %I*:ARRAY[1..64] OF UINT;	//8:OP
		
	//TERM7 EL1008 HQ1
	SensInMac				:BOOL;		//DIGIN CH1			Sensore ingresso macinatore
	R5_S2					:BOOL;		//DIGIN CH2			Val1 aperta
	T5_S3					:BOOL;		//DIGIN CH3			Val2 chiusa
	S1_S3					:BOOL;		//DIGIN CH4			Allarme silos1 pieno
	T6_S1					:BOOL;		//DIGIN CH5			Rotaz catena IFS289
	HQ1_Auto_ON				:BOOL;		//DIGIN CH6			Modo auto-man
	HQ1_P1					:BOOL;		//DIGIN CH7			Reset Allarme
	HQ1_K1					:BOOL;		//DIGIN CH8			---
	
	//TERM8 EL1008 HQ1
	HQ1_MacinatoreON		:BOOL;		//DIGIN CH1 		DA QUADRO MACINATORE
	HQ1_ScorniciatriceON	:BOOL;		//DIGIN CH9 		DA QUADRO SILOS 1
	HQ1_AspirazioneON		:BOOL; 		//DIGIN CH10		DA QUADRO SILOS 1
	I_Fdbk_Km_Area_Nastri_Macinatore : BOOL;
	I_Fdbk_Km_Area_Macinatore:BOOL;		//DIGIN CH11 		feedback contattore area macinatore
	HQ1_BricchettatriceON	:BOOL;		//DIGIN CH6
	
	//TERM9 EL2008 HQ1
//	S1_U1					:BOOL;		//DIGOUT CH1		Valvola aria pulizia ingresso M12
	Dis_Scarico_Hundegger	:BOOL;		//DIGOUT CH1		abilitazione scarico Hundegger	
	HQ1_T1_KA1				:BOOL;		//DIGOUT CH2		T1 Vibrotrasp buca
	HQ1_T2_KA2				:BOOL;		//DIGOUT CH3		T2 Nastro elev buca
	HQ1_T3_KA3				:BOOL;		//DIGOUT CH4		T3 Vibrotrasp macinatore
	HQ1_T5M2_A_KA4			:BOOL;		//DIGOUT CH5		Apre scarico trasp orizz
	HQ1_T5_KA5				:BOOL;		//DIGOUT CH6		Trasp elevat a parete
	HQ1_T6_KA6				:BOOL;		//DIGOUT CH7		Trasp orizza a parete
	HQ1_T5M2_C_KA7			:BOOL;		//DIGOUT CH8		Chiude scarico trasp orizz
		
	//TERM10 EL2008 HQ1
	HQ1_T7_A_KA8			:BOOL;		//DIGOUT CH1		Caricatore macinat Avanti
	HQ1_T7_I_KA9			:BOOL;		//DIGOUT CH2		Caricatore macinat Indietro
	HQ1_M_ON				:BOOL;		//DIGOUT CH3		Macinatore ON
	HQ1_M_OFF				:BOOL;		//DIGOUT CH4		Macinatore OFF		
	HQ1_T4_KA4				:BOOL;		//DIGOUT CH5		T4 Trasportatore da silos a macinatore
	HQ1_S1_ValvolaStellare	:BOOL;		//DIGOUT CH6		Valvola stellare silos 1: AVVIATO DA QUADRO SILOS
	HQ1_RaclaON				:BOOL;		//DIGOUT CH7		Racia :AVVIATO DA QUADRO SILOS
	HQ1_BrichettatriceON	:BOOL;		//DIGOUT CH8		Brichettatrice:AVVIATA DA QUADRO SILOS

	//TERM11 EL3012 HQ1
	T3_S1					:INT;		//ANALOGIN CH1		Pres materiale Ingresso a T3
	T3_S2					:INT;		//ANALOGIN CH2		Pres materiale Uscita da T3
	
	//TERM12 EL3012 HQ1
	S2_S1					:INT;		//ANALOGIN CH1		Liv silos2 UMT 30-6000
	
	//BARRIERA MACINATORE
	I_Barriera_Macinatore	: BOOL;
	
(*****************************************************************)	
(*****************************************************************)	
(*****************************************************************)	
	
	S1_S1					:BOOL;
	S1_S2					:BOOL;		//QUADRO SILOS1		Sensore dig. troppopieno
	
	
	
	
(*****************************************************************)	
(*****************************************************************)	
(*****************************************************************)	
	
	//CIABATTA MCS1
	glo_dig_in_MCS1			AT %I*:ARRAY[1..64] OF BOOL;
	glo_dig_out_MCS1		AT %Q*:ARRAY[1..64] OF BOOL;	
	glo_analog_in_MCS1		AT %I*:ARRAY[1..64] OF INT;	
	glo_analog_out_MCS1		AT %Q*:ARRAY[1..64] OF USINT;	
	glo_WcState_MCS1		AT %I*:ARRAY[1..64] OF BOOL;	//0:Valid, 1:Invalid
	glo_State_MCS1			AT %I*:ARRAY[1..64] OF UINT;	//8:OP
	glo_IOLState_MCS1		AT %I*:ARRAY[1..64] OF USINT;	//3:OP
	
	//BOX16 EP6228-0022 MCS1
	T1_SO1					:INT;		//IOLINK CH1		Pres mat T1, da inizio vibro fino sopra nastro  O1D120
	
	
	
	
(*****************************************************************)	
(*****************************************************************)	
(*****************************************************************)	
	
	//CIABATTA T3C01
	glo_dig_in_T3C01		AT %I*:ARRAY[1..64] OF BOOL;
	glo_dig_out_T3C01		AT %Q*:ARRAY[1..64] OF BOOL;	
	glo_analog_in_T3C01		AT %I*:ARRAY[1..64] OF INT;	
	glo_analog_out_T3C01	AT %Q*:ARRAY[1..64] OF USINT;	
	glo_WcState_T3C01		AT %I*:ARRAY[1..64] OF BOOL;	//0:Valid, 1:Invalid
	glo_State_T3C01			AT %I*:ARRAY[1..64] OF UINT;	//8:OP
	glo_IOLState_T3C01		AT %I*:ARRAY[1..64] OF USINT;	//3:OP

	//BOX17 EP6228-0022 T3C01
	S1_SO2					:INT;			//IOLINK CH2		LIV AVVIO VALV STELLARE UGT514
	S1_PO1					:ES_S1PO1;		//IOLINK CH3		PULSANTIERA BNI005N
	M_PO1					:ES_MPO1;		//IOLINK CH4		PULSANTIERA BNI005M
	S1_Se1					:ES_SEMAFORO;	//IOLINK CH5		SEMAFORO DV2530
	M_Se1					:INT;			//IOLINK CH6		SEMAFORO DV2530	
	T5_S1					:BOOL;			//DIGIN  CH7		ROTAZ CATENA IFS289
	T5_SO1					:INT;			//IOLINK CH8		LIV SCARICO MAC UGT525
	I_Pls_Start_Vibro_Hdd	:BOOL;
	
	
	
(*****************************************************************)	
(*****************************************************************)	
(*****************************************************************)	

	//TWINSAFE
	TS_ErrAck				AT %Q*:BOOL;	//ERRORE ACK
	TS_Run_GrpES			AT %Q*:BOOL;	//RUN Gruppo TwinSAFE EVACUAZIONE SCARTI
	TS_ComErr				AT %I*:BOOL;
	TS_FBErr				AT %I*:BOOL;
	
	TS_AreaM_ON				AT %I*:BOOL;	//STATO AREA MACINATORE
	TS_MPO1_Rst_Area_Macinatore	AT %Q*:BOOL;	//RESET AREA MACINATORE


	TS_AreaS_ON				AT %I*:BOOL;	//STATO AREA SILOS
	TS_S1PO1_btn_Emerg		AT %I*:BOOL;	//STATO FUNGO EMERGENZA da TWINSAFE
	TS_S1PO1_btn_R			AT %Q*:BOOL;	//STATO BOTTONE RIARMO a TWINSAFE
	TS_S1PR1_Door			AT %I*:BOOL;	//STATO PORTA MACINATORE da TWINSAFE
	
	TS_AreaM_OFF				AT %I*:BOOL;	
	TS_AreaS_OFF				AT %I*:BOOL;	
	

(*****************************************************************)	
(*****************************************************************)	
(*****************************************************************)	
	
	//Timer per sensore T5_S1 rotazione catena
	tmr_T5_S1				:TON;
	
	//Logica Aspirazione ON
	LogicaAspirazioneON		:BOOL;		
	
	//HMI - VALORI ATTUALI
	glo_ES_ActVal			:ES_ACTVAL;
	
	//Persistenti - NOVRAM
	glo_ES_Config			AT %Q*:ES_PERSISTENT;

	
	
	//AREA MACINATORE	
	
	//HMI - BOTTONI
	bAbilitaPulsatiera		:BOOL;
	AreaM_ON				:BOOL;
	bIsAuto					:BOOL;	
	
	bAbilitaT1T2			:BOOL;
	bAbilitaT3				:BOOL;
	bAbilitaT4				:BOOL;
	
	bT1_ON					:BOOL;
	bT2_ON					:BOOL;
	bT3_ON					:BOOL;	
	bM_ON					:BOOL;
	bT4_ON					:BOOL;
	bMacinatoreStart		:BOOL;
	bMacinatoreStop			:BOOL;
	bT3T5T6DelayStart		:BOOL;
	
	tT3ON_auto				:INT;		//s

	stepT1T2				:INT;
	stepT3					:INT;
	stepT4					:INT;

	descT1T2				:STRING;
	descT3					:STRING;
	descT4					:STRING;
		
	bSIMULAAuto_ON			:BOOL;	
	bSIMULA_out				:BOOL;
	bSIMULA_in				:BOOL;
	bSIMULA_btnM			:BOOL;
	bSIMULA_btnR			:BOOL;
	bSIMULA_btn0			:BOOL;
	bSIMULA_btnT3			:BOOL;
	
	bMAN_SvuotaT1T2T3		:BOOL;
	
	T3_ModoPausaLavoro	:BOOL;
	bT3EnT1PausaLavoro	:BOOL;
	bT3EnT2PausaLavoro	:BOOL;
	M_Cmd_T3			:BOOL;
	T3_Lavoro			:BOOL;
	
	M_Start_Macinatore_Loc:BOOL;
	
	
	
	//AREA SILOS
	AreaS_ON				:BOOL;
	bSIMULA_BrichettatriceON:BOOL;
	bAbilitaPulsatieraS1PO1	:BOOL;
	bSIMULA_btn0silos		:BOOL;
	bSIMULA_btnRsilos		:BOOL;
		
	S1SO2maxTimeavg			:INT:=10;
	T3S1maxTimeavg			:INT:=2;
	T3S2maxTimeavg			:INT:=2;
	T1SO1maxTimeavg			:INT:=2;

	bMAN_SvuotaS1T4			:BOOL;
		
	bAlarmReset				:BOOL;	
	bAllarmeT3				:BOOL;
	bAllarmeT5				:BOOL;
	bAllarmeT6				:BOOL;
	bAllarmeS2S1			:BOOL;
	bAllarmeT5enable		:BOOL;
	bAllarmeT6enable		:BOOL;
	bAllarmeS2S1enable		:BOOL;
	
	bT1SO1pieno				:BOOL;
	bT3S1pieno				:BOOL;
	bT3S2pieno				:BOOL;
	bS1SO2pieno				:BOOL;
	bS2S1pieno				:BOOL;
	
	altMatT3S1				:INT;
	altMatT3S2				:INT;
	altMatS1SO2				:INT;
	distMatT1SO1			:INT;
	
	glo_ES_ActVal_T1_SO1	:INT;
	sogliaT3S1				:INT;
	sogliaT3S2				:INT;
	sogliaS1SO2				:INT;
	solgiaT1SO1				:INT;
	sogliaS2S1				:INT;
	
END_VAR

// ---- GVLs/RULLI CENTRO TAGLI/GVL_CT_IO.TcGVL
{attribute 'Tc2GvlVarNames'}
VAR_GLOBAL
	
(*****************************************************************)	
//				counicazione Valmec
	Com_delta_1			AT %IW10: INT;
	I_Act_Larghezza_Trave_R1		:INT;


(*****************************************************************)	
	//IO TERMINALE 40 C1CO1
	glo_dig_in_Term_40		AT %I*:ARRAY[1..64] OF BOOL;

	I_Fdbk1_Km_Eme_Zona_1		:BOOL;
	I_Fdbk2_Km_Eme_Zona_1		:BOOL;
	
	I_Fdbk1_Km_Eme_Zona_2		:BOOL;
	I_Fdbk2_Km_Eme_Zona_2		:BOOL;
(*****************************************************************)	
(*****************************************************************)	
(*****************************************************************)	

(*****************************************************************)	
(*****************************************************************)	
(*****************************************************************)	
	//CIABATTA C1CO1
	glo_dig_in_C1CO1		AT %I*:ARRAY[1..64] OF BOOL;
	glo_dig_out_C1CO1		AT %Q*:ARRAY[1..64] OF BOOL;	
	glo_WcState_C1C01		AT %I*:ARRAY[1..64] OF BOOL;	//0:Valid, 1:Invalid
	glo_State_C1C01 		AT %I*:ARRAY[1..64] OF UINT;	//8:OP
	glo_IOLState_C1C01		AT %I*:ARRAY[1..64] OF USINT;	//3:OP

		
	C1CO1_Ev1_Soffio_Px				:BOOL;			//DIGOUT CH0			ev soffio sensori catenaria 1
	C1CO1_Ev2_Soffio_Px				:BOOL;			//DIGOUT CH1			ev soffio sensori catenaria 1
	C1CO1_Ev3_Soffio_Px				:BOOL;			//DIGOUT CH2			ev soffio sensori catenaria 1
	C1CO1_Ventola_Motore_C1M3_Rotaz_C1:BOOL;		//DIGOUT CH3			ventola motore
	
(*****************************************************************)	
(*****************************************************************)	
(*****************************************************************)	
	//CIABATTA C1CO2
	glo_dig_in_C1CO2		AT %I*:ARRAY[1..64] OF BOOL;
	glo_dig_out_C1CO2		AT %Q*:ARRAY[1..64] OF BOOL;	
	glo_WcState_C1C02		AT %I*:ARRAY[1..64] OF BOOL;	//0:Valid, 1:Invalid
	glo_State_C1C02 		AT %I*:ARRAY[1..64] OF UINT;	//8:OP
	glo_IOLState_C1C02		AT %I*:ARRAY[1..64] OF USINT;	//3:OP

		
	C1CO2_Ventola_C1M1_Solleva_C1				:BOOL;			//DIGOUT CH0			ev venbtola raffreddamento
	C1CO2_Ventola_C1M2_Ribalta_C1				:BOOL;			//DIGOUT CH1			ev venbtola raffreddamento

(*****************************************************************)	
(*****************************************************************)	
(*****************************************************************)	
	//CIABATTA C1CD1
	glo_dig_in_C1CD1		AT %I*:ARRAY[1..64] OF BOOL;
	glo_dig_out_C1CD1		AT %Q*:ARRAY[1..64] OF BOOL;	
	glo_analog_in_C1CD1		AT %I*:ARRAY[1..64] OF INT;	
	glo_analog_out_C1CD1	AT %Q*:ARRAY[1..64] OF USINT;	
	glo_WcState_C1CD1		AT %I*:ARRAY[1..64] OF BOOL;	//0:Valid, 1:Invalid
	glo_State_C1CD1 		AT %I*:ARRAY[1..64] OF UINT;	//8:OP
	glo_IOLState_C1CD1		AT %I*:ARRAY[1..64] OF USINT;	//3:OP

		
	C1_Ftc1_Fila4_Presenza		:BOOL;		//DIGIN CH0			fotocellula presenza trave
	C1_Ftc2_Fila4_Presenza		:BOOL;		//DIGIN CH1			fotocellula presenza trave
	C1_Ftc3_Fila4_Presenza		:BOOL;		//DIGIN CH2			fotocellula presenza trave
	C1_Ftc1_Fila3_Presenza		:BOOL;		//DIGIN CH3			fotocellula presenza trave
	C1_Ftc1_Fila1_Presenza		:BOOL;		//DIGIN CH4			fotocellula presenza trave
	C1_Ftc1_Fila2_Presenza		:BOOL;		//DIGIN CH5			fotocellula presenza trave
	C1_Ftc2_Fila1_Presenza		:BOOL;		//DIGIN CH6			fotocellula presenza trave
	C1_Ftc2_Fila3_Presenza		:BOOL;		//DIGIN CH7			fotocellula presenza trave
	
	
(*****************************************************************)	
(*****************************************************************)	
(*****************************************************************)	
	//CIABATTA C1CD2
	glo_dig_in_C1CD2		AT %I*:ARRAY[1..64] OF BOOL;
	glo_dig_out_C1CD2		AT %Q*:ARRAY[1..64] OF BOOL;	
	glo_analog_in_C1CD2		AT %I*:ARRAY[1..64] OF INT;	
	glo_analog_out_C1CD2	AT %Q*:ARRAY[1..64] OF USINT;	
	glo_WcState_C1CD2		AT %I*:ARRAY[1..64] OF BOOL;	//0:Valid, 1:Invalid
	glo_State_C1CD2 		AT %I*:ARRAY[1..64] OF UINT;	//8:OP
	glo_IOLState_C1CD2		AT %I*:ARRAY[1..64] OF USINT;	//3:OP

	
	C1_Ftc3_Fila1_Presenza		:BOOL;		//DIGIN CH0			fotocellula presenza trave
	C1_Ftc3_Fila3_Presenza		:BOOL;		//DIGIN CH1			fotocellula presenza trave
	C1_Ftc2_Fila2_Presenza		:BOOL;		//DIGIN CH2			fotocellula presenza trave
	C1_Ftc4_Fila4_Presenza		:BOOL;		//DIGIN CH3			fotocellula presenza trave
	C1_Ftc3_Fila2_Presenza		:BOOL;		//DIGIN CH4			fotocellula presenza trave
	C1_Ftc5_Fila4_Presenza		:BOOL;		//DIGIN CH5			fotocellula presenza trave
	C1_Ftc4_Fila3_Presenza		:BOOL;		//DIGIN CH6			fotocellula presenza trave
	C1_Ftc4_Fila2_Presenza		:BOOL;		//DIGIN CH7			fotocellula presenza trave

	
(*****************************************************************)	
(*****************************************************************)	
(*****************************************************************)	
	//CIABATTA C1CD3
	glo_dig_in_C1CD3		AT %I*:ARRAY[1..64] OF BOOL;
	glo_dig_out_C1CD3		AT %Q*:ARRAY[1..64] OF BOOL;	
	glo_analog_in_C1CD3		AT %I*:ARRAY[1..64] OF INT;	
	glo_analog_out_C1CD3	AT %Q*:ARRAY[1..64] OF USINT;	
	glo_WcState_C1CD3		AT %I*:ARRAY[1..64] OF BOOL;	//0:Valid, 1:Invalid
	glo_State_C1CD3 		AT %I*:ARRAY[1..64] OF UINT;	//8:OP
	glo_IOLState_C1CD3		AT %I*:ARRAY[1..64] OF USINT;	//3:OP

	
	C1_Ftc7_Fila4_Presenza		:BOOL;		//DIGIN CH0			fotocellula presenza trave
	C1_Ftc6_Fila1_Presenza		:BOOL;		//DIGIN CH1			fotocellula presenza trave
	C1_Ftc6_Fila3_Presenza		:BOOL;		//DIGIN CH2			fotocellula presenza trave
	C1_Ftc6_Fila2_Presenza		:BOOL;		//DIGIN CH3			fotocellula presenza trave
	C1_Ftc6_Fila4_Presenza		:BOOL;		//DIGIN CH4			fotocellula presenza trave
	C1_Ftc5_Fila3_Presenza		:BOOL;		//DIGIN CH5			fotocellula presenza trave
	C1_Ftc5_Fila2_Presenza		:BOOL;		//DIGIN CH6			fotocellula presenza trave
	C1_Ftc4_Fila1_Presenza		:BOOL;		//DIGIN CH7			fotocellula presenza trave		
	

(*****************************************************************)	
(*****************************************************************)	
(*****************************************************************)	
	//CIABATTA C1CD4
	glo_dig_in_C1CD4		AT %I*:ARRAY[1..64] OF BOOL;
	glo_dig_out_C1CD4		AT %Q*:ARRAY[1..64] OF BOOL;	
	glo_analog_in_C1CD4		AT %I*:ARRAY[1..64] OF INT;	
	glo_analog_out_C1CD4	AT %Q*:ARRAY[1..64] OF USINT;	
	glo_WcState_C1CD4		AT %I*:ARRAY[1..64] OF BOOL;	//0:Valid, 1:Invalid
	glo_State_C1CD4 		AT %I*:ARRAY[1..64] OF UINT;	//8:OP
	glo_IOLState_C1CD4		AT %I*:ARRAY[1..64] OF USINT;	//3:OP
	
	
	
	C1_Px_Catena_DW 		:BOOL;		//DIGIN CH0			fotocellula presenza trave
	C1_Px_Catena_UP 		:BOOL;		//DIGIN CH1			fotocellula presenza trave
	C1_Px1_Rotaz_In_Piano  	:BOOL;		//DIGIN CH2			fotocellula presenza trave
	C1_Px2_Rotaz_In_Piano	:BOOL;		//DIGIN CH3			fotocellula presenza trave
	C1_Ftc5_Fila1_Presenza	:BOOL;		//DIGIN CH4			fotocellula presenza trave
	C1_Ftc_Pres_Pz_Da_Hundegger : BOOL;	//DIGIN CH7			fotocellula pezzo in arrivo da Hundegger
	
(*****************************************************************)	
(*****************************************************************)	
(*****************************************************************)	
	//CIABATTA C2CD1
	glo_dig_in_C2CD1		AT %I*:ARRAY[1..64] OF BOOL;
	glo_dig_out_C2CD1		AT %Q*:ARRAY[1..64] OF BOOL;	
	glo_analog_in_C2CD1		AT %I*:ARRAY[1..64] OF INT;	
	glo_analog_out_C2CD1	AT %Q*:ARRAY[1..64] OF USINT;	
	glo_WcState_C2CD1		AT %I*:ARRAY[1..64] OF BOOL;	//0:Valid, 1:Invalid
	glo_State_C2CD1 		AT %I*:ARRAY[1..64] OF UINT;	//8:OP
	glo_IOLState_C2CD1		AT %I*:ARRAY[1..64] OF USINT;	//3:OP

	
	C2_Ftc1_Fila1_Presenza		:BOOL;		//DIGIN CH0			fotocellula presenza trave
	C2_Ftc1_Fila2_Presenza		:BOOL;		//DIGIN CH1			fotocellula presenza trave
	C2_Ftc1_Fila3_Presenza		:BOOL;		//DIGIN CH2			fotocellula presenza trave
	C2_Ftc1_Fila4_Presenza		:BOOL;		//DIGIN CH3			fotocellula presenza trave
	C2_Ftc2_Fila4_Presenza		:BOOL;		//DIGIN CH4			fotocellula presenza trave
	C2_Ftc2_Fila3_Presenza		:BOOL;		//DIGIN CH5			fotocellula presenza trave
	C2_Ftc2_Fila2_Presenza		:BOOL;		//DIGIN CH6			fotocellula presenza trave
	C2_Ftc2_Fila1_Presenza		:BOOL;		//DIGIN CH7			fotocellula presenza trave	

	
(*****************************************************************)	
(*****************************************************************)	
(*****************************************************************)	
	//CIABATTA C2CD2
	glo_dig_in_C2CD2		AT %I*:ARRAY[1..64] OF BOOL;
	glo_dig_out_C2CD2		AT %Q*:ARRAY[1..64] OF BOOL;	
	glo_analog_in_C2CD2		AT %I*:ARRAY[1..64] OF INT;	
	glo_analog_out_C2CD2	AT %Q*:ARRAY[1..64] OF USINT;	
	glo_WcState_C2CD2		AT %I*:ARRAY[1..64] OF BOOL;	//0:Valid, 1:Invalid
	glo_State_C2CD2 		AT %I*:ARRAY[1..64] OF UINT;	//8:OP
	glo_IOLState_C2CD2		AT %I*:ARRAY[1..64] OF USINT;	//3:OP
	
	
	C2_Ftc3_Fila4_Presenza		:BOOL;		//DIGIN CH0			fotocellula presenza trave
	C2_Ftc3_Fila3_Presenza		:BOOL;		//DIGIN CH1			fotocellula presenza trave
	C2_Ftc3_Fila2_Presenza		:BOOL;		//DIGIN CH2			fotocellula presenza trave
	C2_Ftc3_Fila1_Presenza		:BOOL;		//DIGIN CH3			fotocellula presenza trave
	C2_Ftc4_Fila4_Presenza		:BOOL;		//DIGIN CH4			fotocellula presenza trave
	C2_Ftc4_Fila3_Presenza		:BOOL;		//DIGIN CH5			fotocellula presenza trave
	C2_Ftc4_Fila2_Presenza		:BOOL;		//DIGIN CH6			fotocellula presenza trave
	C2_Ftc4_Fila1_Presenza		:BOOL;		//DIGIN CH7			fotocellula presenza trave	
	
	
(*****************************************************************)	
(*****************************************************************)	
(*****************************************************************)	
	//CIABATTA C2CD3
	glo_dig_in_C2CD3		AT %I*:ARRAY[1..64] OF BOOL;
	glo_dig_out_C2CD3		AT %Q*:ARRAY[1..64] OF BOOL;	
	glo_analog_in_C2CD3		AT %I*:ARRAY[1..64] OF INT;	
	glo_analog_out_C2CD3	AT %Q*:ARRAY[1..64] OF USINT;	
	glo_WcState_C2CD3		AT %I*:ARRAY[1..64] OF BOOL;	//0:Valid, 1:Invalid
	glo_State_C2CD3 		AT %I*:ARRAY[1..64] OF UINT;	//8:OP
	glo_IOLState_C2CD3		AT %I*:ARRAY[1..64] OF USINT;	//3:OP


	C2_Ftc5_Fila4_Presenza		:BOOL;		//DIGIN CH0			fotocellula presenza trave
	C2_Ftc5_Fila3_Presenza		:BOOL;		//DIGIN CH1			fotocellula presenza trave
	C2_Ftc5_Fila2_Presenza		:BOOL;		//DIGIN CH2			fotocellula presenza trave
	C2_Ftc5_Fila1_Presenza		:BOOL;		//DIGIN CH3			fotocellula presenza trave
	C2_Ftc6_Fila4_Presenza		:BOOL;		//DIGIN CH4			fotocellula presenza trave
	C2_Ftc6_Fila3_Presenza		:BOOL;		//DIGIN CH5			fotocellula presenza trave
	C2_Ftc6_Fila2_Presenza		:BOOL;		//DIGIN CH6			fotocellula presenza trave
	C2_Ftc6_Fila1_Presenza		:BOOL;		//DIGIN CH7			fotocellula presenza trave	
	
	
(*****************************************************************)	
(*****************************************************************)	
(*****************************************************************)	
	//CIABATTA C2CD4
	glo_dig_in_C2CD4		AT %I*:ARRAY[1..64] OF BOOL;
	glo_dig_out_C2CD4		AT %Q*:ARRAY[1..64] OF BOOL;	
	glo_analog_in_C2CD4		AT %I*:ARRAY[1..64] OF INT;	
	glo_analog_out_C2CD4	AT %Q*:ARRAY[1..64] OF USINT;	
	glo_WcState_C2CD4		AT %I*:ARRAY[1..64] OF BOOL;	//0:Valid, 1:Invalid
	glo_State_C2CD4 		AT %I*:ARRAY[1..64] OF UINT;	//8:OP
	glo_IOLState_C2CD4		AT %I*:ARRAY[1..64] OF USINT;	//3:OP	
	
	
	C2_Ftc7_Fila4_Presenza		:BOOL;		//DIGIN CH0			fotocellula presenza trave
	C2_Ftc7_Fila3_Presenza		:BOOL;		//DIGIN CH1			fotocellula presenza trave
	C2_Ftc7_Fila2_Presenza		:BOOL;		//DIGIN CH2			fotocellula presenza trave
	C2_Ftc7_Fila1_Presenza		:BOOL;		//DIGIN CH3			fotocellula presenza trave
	R1_Px_Rulliera_UP   		:BOOL;		//DIGIN CH4			proximity rulliera alta
	R1_Px_Rulliera_DW			:BOOL;		//DIGIN CH5			proximity rulliera bassa
		

(*****************************************************************)	
(*****************************************************************)	
(*****************************************************************)	
	//CIABATTA C2CO1
	glo_dig_in_C2CO1		AT %I*:ARRAY[1..64] OF BOOL;
	glo_dig_out_C2CO1		AT %Q*:ARRAY[1..64] OF BOOL;	
	glo_WcState_C2C01		AT %I*:ARRAY[1..64] OF BOOL;	//0:Valid, 1:Invalid
	glo_State_C2C01 		AT %I*:ARRAY[1..64] OF UINT;	//8:OP
	glo_IOLState_C2C01		AT %I*:ARRAY[1..64] OF USINT;	//3:OP

	C2CO1_Ev1_Soffio_Px				:BOOL;			//DIGOUT CH1			ev soffio sensori catenaria 2
	C2CO1_Ev2_Soffio_Px				:BOOL;			//DIGOUT CH2			ev soffio sensori catenaria 2
	C2CO1_Ev3_Soffio_Px				:BOOL;			//DIGOUT CH3			ev soffio sensori catenaria 2
	C2CO1_Ventola_Motore_C2M1_Rotaz_C2:BOOL;			//DIGOUT CH4			ev venbtola raffreddamento
	C2CO1_Ventola_R1M2_Rotaz_R2		:BOOL;			//DIGOUT CH5			ev venbtola raffreddamento

		
(*****************************************************************)	
(*****************************************************************)	
(*****************************************************************)	
	//CIABATTA C2CO2
	glo_dig_in_C2CO2		AT %I*:ARRAY[1..64] OF BOOL;
	glo_dig_out_C2CO2		AT %Q*:ARRAY[1..64] OF BOOL;	
	glo_WcState_C2CO2		AT %I*:ARRAY[1..64] OF BOOL;	//0:Valid, 1:Invalid
	glo_State_C2CO2 		AT %I*:ARRAY[1..64] OF UINT;	//8:OP
	glo_IOLState_C2CO2		AT %I*:ARRAY[1..64] OF USINT;	//3:OP	
	
	
	
	//PULSANTIERA C1P1
	glo_dig_in_C1P1			AT %I*:ARRAY[1..64] OF BOOL;
	glo_dig_out_C1P1		AT %Q*:ARRAY[1..64] OF BOOL;	

	C1P1_Pls_Marcia		:BOOL;		//DIGIN CH1			pulsante marcia
	C1P1_Rst_Eme		:BOOL;		//DIGIN CH2			pulsante ripristino emergenza

	C1P1_Pls_C1_Fw		:BOOL;		//DIGIN CH3			pulsante comando discesa rulliera 1
	C1P1_Pls_C1_Bk		:BOOL;		//DIGIN CH4			pulsante comando discesa rulliera 1
	C1P1_Pls_C1_Dw		:BOOL;		//DIGIN CH5			pulsante comando discesa rulliera 1
	C1P1_Pls_C1_Up		:BOOL;		//DIGIN CH6			pulsante comando salita rulliera 1
	
	C1P1_Pls_C1_Rot_Fw	:BOOL;		//DIGIN CH7			pulsante comando discesa rulliera 1
	C1P1_Pls_C1_Rot_Bk	:BOOL;		//DIGIN CH8			pulsante comando salita rulliera 1
	
	C1P1_Lp_Eme_Ok		:BOOL;		//DIGOUT CH9		pulsante comando salita rulliera 1
	C1P1_Lp_Marcia_On	:BOOL;		//DIGOUT CH10		pulsante comando salita rulliera 1

	
	//PULSANTIERA R1P1
	glo_dig_in_R1P1			AT %I*:ARRAY[1..64] OF BOOL;	
	glo_dig_out_R1P1		AT %Q*:ARRAY[1..64] OF BOOL;	

	R1P1_Sel_Chiave		:BOOL;		//DIGIN CH1			selettore a chiave
	R1P1_Pls_Marcia		:BOOL;		//DIGIN CH2			pulsante marcia
	R1P1_Rst_Eme		:BOOL;		//DIGIN CH3			pulsante ripristino emergenza

	R1P1_Pls_C2_Fw		:BOOL;		//DIGIN CH4			pulsante comando discesa rulliera 1
	R1P1_Pls_C2_Bk		:BOOL;		//DIGIN CH5			pulsante comando discesa rulliera 1

	R1P1_Pls_R1_Fw		:BOOL;		//DIGIN CH6			pulsante comando discesa rulliera 1
	R1P1_Pls_R1_Bk		:BOOL;		//DIGIN CH7			pulsante comando discesa rulliera 1
	R1P1_Pls_R1_Dw		:BOOL;		//DIGIN CH8			pulsante comando discesa rulliera 1
	R1P1_Pls_R1_Up		:BOOL;		//DIGIN CH9			pulsante comando salita rulliera 1
	
	R1P1_Lp_Eme_Ok		:BOOL;		//DIGOUT CH10			pulsante comando salita rulliera 1
	R1P1_Lp_Marcia_On	:BOOL;		//DIGOUT CH11		pulsante comando salita rulliera 1
	
	
	//PULSANTIERA R1P2
	glo_dig_in_R1P2			AT %I*:ARRAY[1..64] OF BOOL;	
	glo_dig_out_R1P2		AT %Q*:ARRAY[1..64] OF BOOL;	

	R1P2_Pls_Ciclo_Singolo	:BOOL;		//DIGIN CH1			pulsante richiesta ciclo singolo rulliera R1
	R1P2_Pls_Ciclo_Continuo	:BOOL;		//DIGIN CH2			pulsante richiesta ciclo continuo rulliera R1
	R1P2_Pls_Marcia			:BOOL;
	R1P2_Pls_Marcia_Off		:BOOL;
	
	//PULSANTIERA R1P3
	glo_dig_in_R1P3			AT %I*:ARRAY[1..64] OF BOOL;	
	glo_dig_out_R1P3		AT %Q*:ARRAY[1..64] OF BOOL;	

	R1P3_Pls_Ciclo_Singolo	:BOOL;		//DIGIN CH1			pulsante richiesta ciclo singolo rulliera R1
	R1P3_Pls_Ciclo_Continuo	:BOOL;		//DIGIN CH2			pulsante richiesta ciclo continuo rulliera R1
	R1P3_Pls_Marcia			:BOOL;
	R1P3_Pls_Marcia_Off		:BOOL;

	//PULSANTIERA R1P4
	glo_dig_in_R1P4			AT %I*:ARRAY[1..64] OF BOOL;	
	glo_dig_out_R1P4		AT %Q*:ARRAY[1..64] OF BOOL;	

	R1P4_Pls_Ciclo_Singolo	:BOOL;		//DIGIN CH1			pulsante richiesta ciclo singolo rulliera R1
	R1P4_Pls_Ciclo_Continuo	:BOOL;		//DIGIN CH2			pulsante richiesta ciclo continuo rulliera R1
	R1P4_Pls_Marcia			:BOOL;
	R1P4_Pls_Marcia_Off		:BOOL;
	
	
	//PULSANTIERA R1P5
	glo_dig_in_R1P5			AT %I*:ARRAY[1..64] OF BOOL;	
	glo_dig_out_R1P5		AT %Q*:ARRAY[1..64] OF BOOL;	

	R1P5_Pls_Ciclo_Singolo	:BOOL;		//DIGIN CH1			pulsante richiesta ciclo singolo rulliera R1
	R1P5_Pls_Ciclo_Continuo	:BOOL;		//DIGIN CH2			pulsante richiesta ciclo continuo rulliera R1
	R1P5_Pls_Marcia			:BOOL;
	R1P5_Pls_Marcia_Off		:BOOL;
	
	
	//PULSANTIERA R1P6
	glo_dig_in_R1P6			AT %I*:ARRAY[1..64] OF BOOL;	
	glo_dig_out_R1P6		AT %Q*:ARRAY[1..64] OF BOOL;	

	R1P6_Pls_Ciclo_Singolo	:BOOL;		//DIGIN CH1			pulsante richiesta ciclo singolo rulliera R1
	R1P6_Pls_Ciclo_Continuo	:BOOL;		//DIGIN CH2			pulsante richiesta ciclo continuo rulliera R1
	R1P6_Pls_Marcia			:BOOL;
	R1P6_Pls_Marcia_Off		:BOOL;


	//SEMAFORO
	RCT_Semaforo					:ES_SEMAFORO;	//IOLINK CH5		SEMAFORO DV2530

	//colori
	// 1 blu
	// 2 verde
	// 3 azzurro
	// 4 rosso
	// 5 violetto
	// 6 arancione
	
	RCT_Semaforo_Led_1			:USINT;				//led 1 il piu in basso
	RCT_Semaforo_Led_2			:USINT;				//led 1 il piu in basso
	RCT_Semaforo_Led_3			:USINT;				//led 1 il piu in basso
	RCT_Semaforo_Led_4			:USINT;				//led 1 il piu in basso
	RCT_Semaforo_Led_5			:USINT;				//led 1 il piu in basso

(*****************************************************************)	
(*****************************************************************)	
(*****************************************************************)	
	//CIABATTA C3CD1
	glo_dig_in_C3CD1		AT %I*:ARRAY[1..64] OF BOOL;
	glo_dig_out_C3CD1		AT %Q*:ARRAY[1..64] OF BOOL;	
	glo_WcState_C3CD1		AT %I*:ARRAY[1..64] OF BOOL;	//0:Valid, 1:Invalid
	glo_State_C3CD1 		AT %I*:ARRAY[1..64] OF UINT;	//8:OP
	glo_IOLState_C3CD1		AT %I*:ARRAY[1..64] OF USINT;	//3:OP


	C4_Ftc4_Presenza_Ingresso		:BOOL;		//DIGIN CH0			fotocellula presenza trave
	C4_Ftc5_Presenza_Ingresso		:BOOL;		//DIGIN CH0			fotocellula presenza trave
	C4_Ftc6_Presenza_Ingresso		:BOOL;		//DIGIN CH0			fotocellula presenza trave
	C4_Ftc7_Presenza_Ingresso		:BOOL;		//DIGIN CH0			fotocellula presenza trave
	C4_Ftc4_Presenza_Uscita			:BOOL;		//DIGIN CH0			fotocellula presenza trave
	C4_Ftc5_Presenza_Uscita			:BOOL;		//DIGIN CH0			fotocellula presenza trave
	C4_Ftc6_Presenza_Uscita			:BOOL;		//DIGIN CH0			fotocellula presenza trave
	C4_Ftc7_Presenza_Uscita			:BOOL;		//DIGIN CH0			fotocellula presenza trave
		
(*****************************************************************)	
(*****************************************************************)	
(*****************************************************************)	
	//CIABATTA C3CD2
	glo_dig_in_C3CD2		AT %I*:ARRAY[1..64] OF BOOL;
	glo_dig_out_C3CD2		AT %Q*:ARRAY[1..64] OF BOOL;	
	glo_WcState_C3CD2		AT %I*:ARRAY[1..64] OF BOOL;	//0:Valid, 1:Invalid
	glo_State_C3CD2			AT %I*:ARRAY[1..64] OF UINT;	//8:OP
	glo_IOLState_C3CD2		AT %I*:ARRAY[1..64] OF USINT;	//3:OP
	
	
	C4_Ftc1_Presenza_Ingresso		:BOOL;		//DIGIN CH0			fotocellula presenza trave
	C4_Ftc2_Presenza_Ingresso		:BOOL;		//DIGIN CH0			fotocellula presenza trave
	C4_Ftc3_Presenza_Ingresso		:BOOL;		//DIGIN CH0			fotocellula presenza trave
	C4_Ftc1_Presenza_Uscita			:BOOL;		//DIGIN CH0			fotocellula presenza trave
	C4_Ftc2_Presenza_Uscita			:BOOL;		//DIGIN CH0			fotocellula presenza trave
	C4_Ftc3_Presenza_Uscita			:BOOL;		//DIGIN CH0			fotocellula presenza trave
	
	
(*****************************************************************)	
(*****************************************************************)	
(*****************************************************************)	
	//CIABATTA C3CO1
	glo_dig_in_C3CO1		AT %I*:ARRAY[1..64] OF BOOL;
	glo_dig_out_C3CO1		AT %Q*:ARRAY[1..64] OF BOOL;	
	glo_WcState_C3CO1		AT %I*:ARRAY[1..64] OF BOOL;	//0:Valid, 1:Invalid
	glo_State_C3CO1 		AT %I*:ARRAY[1..64] OF UINT;	//8:OP
	glo_IOLState_C3CO1		AT %I*:ARRAY[1..64] OF USINT;	//3:OP	
	
	
	R2_Paletta_Presenza_Pezzo:BOOL;
	
	//PULSANTIERA C4P1
	glo_dig_in_C4P1			AT %I*:ARRAY[1..64] OF BOOL;
	glo_dig_out_C4P1		AT %Q*:ARRAY[1..64] OF BOOL;		
	
	C4P1_Sel_Chiave		:BOOL;		//DIGIN CH1			selettore a chiave
	C4P1_Pls_Marcia		:BOOL;		//DIGIN CH1			pulsante marcia
	C4P1_Rst_Eme		:BOOL;		//DIGIN CH2			pulsante ripristino emergenza
	
	C4P1_Pls_C3_Fw		:BOOL;		//DIGIN CH3			pulsante comando avanti catenaria 3
	C4P1_Pls_C3_Bk		:BOOL;		//DIGIN CH4			pulsante comando indietro catenaria 3	

	C4P1_Pls_C4_Fw		:BOOL;		//DIGIN CH3			pulsante comando avanti catenaria 4
	C4P1_Pls_C4_Bk		:BOOL;		//DIGIN CH4			pulsante comando indietro catenaria 4	
	
	C4P1_Lp_Eme_Ok		:BOOL;		//DIGOUT CH9		lampada emergenza ok
	C4P1_Lp_Marcia_On	:BOOL;		//DIGOUT CH10		lampoada marcia on		
	
	
	//PULSANTIERA C4PO1
	glo_dig_in_C4PO1			AT %I*:ARRAY[1..64] OF BOOL;
	glo_dig_out_C4PO1		AT %Q*:ARRAY[1..64] OF BOOL;		
	
	C4PO1_Pls_R2_Fw		:BOOL;		//DIGIN CH3			pulsante comando avanti rulliera 2
	C4PO1_Pls_R2_Bk		:BOOL;		//DIGIN CH4			pulsante comando indietro rulliera 2	
	C4PO1_Pls_R2_Dw		:BOOL;		//DIGIN CH5			pulsante comando discesa rulliera 2
	C4PO1_Pls_R2_Up		:BOOL;		//DIGIN CH6			pulsante comando salita rulliera 2
	
	C4PO1_Pls_C5_Fw		:BOOL;		//DIGIN CH3			pulsante comando avanti catenaria 5
	C4PO1_Pls_C5_Bk		:BOOL;		//DIGIN CH4			pulsante comando indietro catenaria 5	
	
	C4PO1_Pls_C6_Fw		:BOOL;		//DIGIN CH3			pulsante comando avanti catenaria 6
	C4PO1_Pls_C6_Bk		:BOOL;		//DIGIN CH4			pulsante comando indietro catenaria 6	

	
	C3CO1_Ev1_Soffio_Px	: BOOL;
	C3CO1_Ev2_Soffio_Px	: BOOL;
(*****************************************************************)	
(*****************************************************************)	
(*****************************************************************)	
	//CIABATTA C5CO1
	glo_dig_in_C5CO1		AT %I*:ARRAY[1..64] OF BOOL;
	glo_dig_out_C5CO1		AT %Q*:ARRAY[1..64] OF BOOL;	
	glo_WcState_C5CO1		AT %I*:ARRAY[1..64] OF BOOL;	//0:Valid, 1:Invalid
	glo_State_C25O21		AT %I*:ARRAY[1..64] OF UINT;	//8:OP
	glo_IOLState_C5CO1		AT %I*:ARRAY[1..64] OF USINT;	//3:OP	

	C5CO1_Ventola_Motore_Rotaz_C3	:BOOL;		//DIGOUT CH3			ventola motore	
	C5CO1_Ventola_Motore_Rotaz_C5	:BOOL;		//DIGOUT CH3			ventola motore
	C5CO1_Ventola_Motore_Rotaz_C6	:BOOL;		//DIGOUT CH3			ventola motore
	
	C5CO1_Ventola_Motore_Rotaz_C4	:BOOL;		//DIGOUT CH3			ventola motore
	
	C5CO1_Ev1_Soffio_Px_C5_C6				:BOOL;			//DIGOUT CH0			ev soffio sensori catenaria 3
	C5CO1_Ev2_Soffio_Px_C5_C6				:BOOL;			//DIGOUT CH1			ev soffio sensori catenaria 3
	C5CO1_Ev3_Soffio_Px_C5_C6				:BOOL;			//DIGOUT CH2			ev soffio sensori catenaria 3

	
(*****************************************************************)	
(*****************************************************************)	
(*****************************************************************)	
	//CIABATTA C5CO2
	glo_dig_in_C5CO2		AT %I*:ARRAY[1..64] OF BOOL;
	glo_dig_out_C5CO2		AT %Q*:ARRAY[1..64] OF BOOL;	
	glo_WcState_C5CO2		AT %I*:ARRAY[1..64] OF BOOL;	//0:Valid, 1:Invalid
	glo_State_C25O2 		AT %I*:ARRAY[1..64] OF UINT;	//8:OP
	glo_IOLState_C5CO2		AT %I*:ARRAY[1..64] OF USINT;	//3:OP	
	
	
	R3_Paletta_Presenza_Pezzo:BOOL;
	
	//PULSANTIERA R3P1
	glo_dig_in_R3P1			AT %I*:ARRAY[1..64] OF BOOL;
	glo_dig_out_R3P1		AT %Q*:ARRAY[1..64] OF BOOL;	
	
	R3P1_Pls_Singolo	:BOOL;
	R3P1_Pls_Marcia		:BOOL;
	R3P1_Pls_Infinito	:BOOL;
	
	
	//PULSANTIERA R3P2
	glo_dig_in_R3P2			AT %I*:ARRAY[1..64] OF BOOL;
	glo_dig_out_R3P2		AT %Q*:ARRAY[1..64] OF BOOL;	
	
	R3P2_Pls_Singolo	:BOOL;
	R3P2_Pls_Marcia		:BOOL;
	R3P2_Pls_Infinito	:BOOL;
	
	
	//PULSANTIERA R3P3
	glo_dig_in_R3P3			AT %I*:ARRAY[1..64] OF BOOL;
	glo_dig_out_R3P3		AT %Q*:ARRAY[1..64] OF BOOL;	

    R3P3_Pls_Singolo	:BOOL;
	R3P3_Pls_Marcia		:BOOL;
	R3P3_Pls_Infinito	:BOOL;

	
	//PULSANTIERA R3P4	
	glo_dig_in_R3P4			AT %I*:ARRAY[1..64] OF BOOL;
	glo_dig_out_R3P4		AT %Q*:ARRAY[1..64] OF BOOL;	

	R3P4_Sel_Chiave		:BOOL;		//DIGIN CH1			selettore a chiave
	R3P4_Pls_Marcia		:BOOL;		//DIGIN CH1			pulsante marcia
	R3P4_Rst_Eme		:BOOL;		//DIGIN CH2			pulsante ripristino emergenza


	R3P4_Pls_C5_Fw		:BOOL;		//DIGIN CH3			pulsante comando avanti catenaria 5
	R3P4_Pls_C5_Bk		:BOOL;		//DIGIN CH4			pulsante comando indietro catenaria 5	

	R3P4_Pls_C6_Fw		:BOOL;		//DIGIN CH3			pulsante comando avanti catenaria 5
	R3P4_Pls_C6_Bk		:BOOL;		//DIGIN CH4			pulsante comando indietro catenaria 5	
		
	R3P4_Pls_R3_Fw		:BOOL;		//DIGIN CH3			pulsante comando avanti rulliera 3
	R3P4_Pls_R3_Bk		:BOOL;		//DIGIN CH4			pulsante comando indietro rulliera 3
	R3P4_Pls_R3_Dw		:BOOL;		//DIGIN CH5			pulsante comando discesa rulliera 3
	R3P4_Pls_R3_Up		:BOOL;		//DIGIN CH6			pulsante comando salita rulliera 3
	
	R3P4_Lp_Eme_Ok		:BOOL;		//DIGOUT CH9		lampada emergenza ok
	R3P4_Lp_Marcia_On	:BOOL;		//DIGOUT CH10		lampoada marcia on		
	
	C5CO2_Ventola_Motore_Rotaz_R3	:BOOL;		//DIGOUT CH3			ventola motore
	C5CO2_Ventola_Motore_Rotaz_R2	:BOOL;		//DIGOUT CH3			ventola motore	
	
	
(*****************************************************************)	
(*****************************************************************)	
(*****************************************************************)	
	//CIABATTA C5CD1
	glo_dig_in_C5CD1		AT %I*:ARRAY[1..64] OF BOOL;
	glo_dig_out_C5CD1		AT %Q*:ARRAY[1..64] OF BOOL;	
	glo_WcState_C5CD1		AT %I*:ARRAY[1..64] OF BOOL;	//0:Valid, 1:Invalid
	glo_State_C25D1 		AT %I*:ARRAY[1..64] OF UINT;	//8:OP
	glo_IOLState_C5CD1		AT %I*:ARRAY[1..64] OF USINT;	//3:OP		

	C5_Ftc1_Presenza		:BOOL;		//DIGIN CH0			fotocellula presenza trave
	C5_Ftc2_Presenza		:BOOL;		//DIGIN CH0			fotocellula presenza trave
	C5_Ftc3_Presenza		:BOOL;		//DIGIN CH0			fotocellula presenza trave
	
	C6_Ftc1_Presenza		:BOOL;		//DIGIN CH0			fotocellula presenza trave
	C6_Ftc2_Presenza		:BOOL;		//DIGIN CH0			fotocellula presenza trave
	C6_Ftc3_Presenza		:BOOL;		//DIGIN CH0			fotocellula presenza trave
	
	R3_Ftc1_Presenza		:BOOL;		//DIGIN CH0			fotocellula presenza trave
	R3_Ftc2_Presenza		:BOOL;		//DIGIN CH0			fotocellula presenza trave
	
		
(*****************************************************************)	
(*****************************************************************)	
(*****************************************************************)	
	//CIABATTA C5CD2
	glo_dig_in_C5CD2		AT %I*:ARRAY[1..64] OF BOOL;
	glo_dig_out_C5CD2		AT %Q*:ARRAY[1..64] OF BOOL;	
	glo_WcState_C5CD2		AT %I*:ARRAY[1..64] OF BOOL;	//0:Valid, 1:Invalid
	glo_State_C25D2 		AT %I*:ARRAY[1..64] OF UINT;	//8:OP
	glo_IOLState_C5CD2		AT %I*:ARRAY[1..64] OF USINT;	//3:OP		
	
	R3_Px_Rulliera_UP		:BOOL;		//DIGIN CH4			proximity rulliera alta
	R3_Px_Rulliera_DW		:BOOL;		//DIGIN CH5			proximity rulliera bassa
	
	C5_Ftc4_Presenza		:BOOL;		//DIGIN CH0			fotocellula presenza trave
	
	C6_Ftc4_Presenza		:BOOL;		//DIGIN CH0			fotocellula presenza trave
	C6_Ftc5_Presenza		:BOOL;		//DIGIN CH0			fotocellula presenza trave
	
	R3_Ftc3_Presenza		:BOOL;		//DIGIN CH0			fotocellula presenza trave
	R3_Ftc4_Presenza		:BOOL;		//DIGIN CH0			fotocellula presenza trave
	R3_Ftc5_Presenza		:BOOL;		//DIGIN CH0			fotocellula presenza trave
	
	
(*****************************************************************)	
(*****************************************************************)	
(*****************************************************************)	
	//CIABATTA C5CD3
	glo_dig_in_C5CD3		AT %I*:ARRAY[1..64] OF BOOL;
	glo_dig_out_C5CD3		AT %Q*:ARRAY[1..64] OF BOOL;	
	glo_WcState_C5CD3		AT %I*:ARRAY[1..64] OF BOOL;	//0:Valid, 1:Invalid
	glo_State_C25D3 		AT %I*:ARRAY[1..64] OF UINT;	//8:OP
	glo_IOLState_C5CD3		AT %I*:ARRAY[1..64] OF USINT;	//3:OP			
	
	
	R2_Px_Rulliera_UP		:BOOL;		//DIGIN CH4			proximity rulliera alta
	R2_Px_Rulliera_DW		:BOOL;		//DIGIN CH5			proximity rulliera bassa
	
	C5_Ftc5_Presenza		:BOOL;		//DIGIN CH0			fotocellula presenza trave
	C5_Ftc6_Presenza		:BOOL;		//DIGIN CH0			fotocellula presenza trave
	
	C6_Ftc6_Presenza		:BOOL;		//DIGIN CH0			fotocellula presenza trave
	C6_Ftc7_Presenza		:BOOL;		//DIGIN CH0			fotocellula presenza trave

	R3_Ftc6_Presenza		:BOOL;		//DIGIN CH0			fotocellula presenza trave
	R3_Ftc7_Presenza		:BOOL;		//DIGIN CH0			fotocellula presenza trave

	C3_Ftc_Pezzo_Scaricato_C5	:BOOL;		//DIGIN CH0			fotocellula presenza trave
		
	R2_Px_Presenza_Pezzo	:BOOL;		//DIGIN CH0			paletta presenza trave
	
	R1_Paletta_Presenza_Pezzo:BOOL;

	
(*****************************************************************)	
(*****************************************************************)	
(*****************************************************************)	
	//SAFETY C2_CS1
	glo_dig_in_C2_CS1		AT %I*:ARRAY[1..8] OF BOOL;
	glo_dig_out_C2_CS1		AT %Q*:ARRAY[1..8] OF BOOL;	
	glo_WcState_C2_CS1		AT %I*:ARRAY[1..8] OF BOOL;	//0:Valid, 1:Invalid
	glo_State_C2_CS1 		AT %I*:ARRAY[1..8] OF UINT;	//8:OP
	glo_IOLState_C2_CS1		AT %I*:ARRAY[1..8] OF USINT;	//3:OP	

	C1P1_Pls_Eme				:BOOL;		//C2_CS1 CH2
	R1P1_Pls_Eme				:BOOL;		//C2_CS1 CH8
	R1P2_Pls_Eme				:BOOL;		//C2_CS1 CH4
	R1P3_Pls_Eme				:BOOL;		//C2_CS2 CH6


	//SAFETY C2_CS2
	glo_dig_in_C2_CS2		AT %I*:ARRAY[1..8] OF BOOL;
	glo_dig_out_C2_CS2		AT %Q*:ARRAY[1..8] OF BOOL;	
	glo_WcState_C2_CS2		AT %I*:ARRAY[1..8] OF BOOL;	//0:Valid, 1:Invalid
	glo_State_C2_CS2 		AT %I*:ARRAY[1..8] OF UINT;	//8:OP
	glo_IOLState_C2_CS2		AT %I*:ARRAY[1..8] OF USINT;	//3:OP

	R1P4_Pls_Eme				:BOOL;		//C2_CS2 CH2
	R1P5_Pls_Eme				:BOOL;		//C2_CS2 CH4
	R1P6_Pls_Eme				:BOOL;		//C2_CS2 CH6
	

	//SAFETY C5_CS1
	glo_dig_in_C5_CS1		AT %I*:ARRAY[1..8] OF BOOL;
	glo_dig_out_C5_CS1		AT %Q*:ARRAY[1..8] OF BOOL;	
	glo_WcState_C5_CS1		AT %I*:ARRAY[1..8] OF BOOL;	//0:Valid, 1:Invalid
	glo_State_C5_CS1		AT %I*:ARRAY[1..8] OF UINT;	//8:OP
	glo_IOLState_C5_CS1		AT %I*:ARRAY[1..8] OF USINT;	//3:OP

	
	R3P4_Pls_Eme				:BOOL;		//C5_CS1 CH8
	R3P1_Pls_Eme				:BOOL;		//C5_CS1 CH2
	R3P2_Pls_Eme				:BOOL;		//C5_CS1 CH4
	R3P3_Pls_Eme				:BOOL;		//C5_CS1 CH6

	
	//SAFETY C3_CS1
	glo_dig_in_C3_CS1		AT %I*:ARRAY[1..8] OF BOOL;
	glo_dig_out_C3_CS1		AT %Q*:ARRAY[1..8] OF BOOL;	
	glo_WcState_C3_CS1		AT %I*:ARRAY[1..8] OF BOOL;	//0:Valid, 1:Invalid
	glo_State_C3_CS1		AT %I*:ARRAY[1..8] OF UINT;	//8:OP
	glo_IOLState_C3_CS1		AT %I*:ARRAY[1..8] OF USINT;	//3:OP
	
	C4P1_Pls_Eme				:BOOL;		//C3_CS1 CH2

	//SAFETY BOX18
	glo_dig_in_BOX18		AT %I*:ARRAY[1..8] OF BOOL;
	glo_dig_out_BOX18		AT %Q*:ARRAY[1..8] OF BOOL;	
	glo_WcState_BOX18		AT %I*:ARRAY[1..8] OF BOOL;	//0:Valid, 1:Invalid
	glo_State_BOX18			AT %I*:ARRAY[1..8] OF UINT;	//8:OP
	glo_IOLState_C3_BOX18		AT %I*:ARRAY[1..8] OF USINT;	//3:OP	
	
	PB_Eme_Macinatore			:BOOL;		//COX18 EP1908 CH2
	
(*****************************************************************)	
(*****************************************************************)	
(*****************************************************************)	
	//plc Valmec
	RD_plc_Valmec		AT %I*:INT;
	WR_plc_Valmec		AT %Q*:INT;	


	WR_Req_Start_Aspirazione	AT %Q*:BYTE;
	RD_Aspirazione_RUN			AT %I*:BYTE;

(*****************************************************************)	
(*****************************************************************)	
(*****************************************************************)	
//ciclo svuotamento Hdd
	PB_Start_Svuotamento_Hundegger			:BOOL;
	I_Macinatore_Run						:BOOL;
(*****************************************************************)	
(*****************************************************************)	
(*****************************************************************)	

	//TWINSAFE

	TS_R1P1_Pls_Eme		AT %I*:BOOL;	//STATO FUNGO EMERGENZA da TWINSAFE
	TS_C1P1_Pls_Eme		AT %I*:BOOL;	//STATO FUNGO EMERGENZA da TWINSAFE

	TS_R1P1_Reset_Eme			AT %Q*:BOOL;	//STATO BOTTONE RIARMO a TWINSAFE
	TS_R1P1_Reset_Eme_2			AT %Q*:BOOL;	//STATO BOTTONE RIARMO a TWINSAFE
	TS_C1P1_Reset_Eme			AT %Q*:BOOL;	//STATO BOTTONE RIARMO a TWINSAFE
	
	
	
	
(*****************************************************************)	
(*****************************************************************)	
(*****************************************************************)		
END_VAR
	

VAR_GLOBAL PERSISTENT
	
	C1_Ciclo_Polmone_Sel					:BOOL;
	C4_Ciclo_Rientro_Man_Sel				:BOOL;
	
	C1_Ribalta_Rot_0_Position				:LREAL;
	C1_Ribalta_Rot_Fw_Position				:LREAL;	
	C1_Ribalta_Rot_Bk_Position				:LREAL;
	
	C1_Solleva_Up_Position					:LREAL;	
	C1_Solleva_Dw_Position					:LREAL;
	C1_Solleva_Dw_Position_Rotaz			:LREAL;
	C1_Solleva_DW_Position_FI_Rotaz			:LREAL;
	
	Catenarie_Acc_Set				: LREAL;
	Catenarie_Dec_Set				: LREAL;
	
	Rulliere_Acc_Set				: LREAL;
	Rulliere_Dec_Set				: LREAL;
	
	R1_Rotazione_Jog_Speed			: LREAL;
	R1_Solleva_Jog_Speed			: WORD;
	C1_Rotazione_Jog_Speed			: LREAL;
	C1_Rotazione_Jog_Speed_2		: LREAL;

	C2_Rotazione_Jog_Speed			: LREAL;
	C2_Rotazione_Jog_Speed_2		: LREAL;
	C1_Ribalta_Jog_Speed			: LREAL;
	C1_Solleva_Jog_Speed			: LREAL;
	
	C3_Rotazione_Jog_Speed			: LREAL;
	C4_Rotazione_Jog_Speed			: LREAL;
	C5_Rotazione_Jog_Speed			: LREAL;
	C6_Rotazione_Jog_Speed			: LREAL;
	
	R3_Rotazione_Jog_Speed			: LREAL;
	R3_Solleva_Jog_Speed			: WORD;
	
	R2_Rotazione_Jog_Speed			: LREAL;
	R2_Solleva_Jog_Speed			: WORD;
	


	Ribaltamento_C1_Quota_Preset_Enc	:LREAL;
	Sollevamento_C1_Quota_Preset_Enc	:LREAL;
	
	Catenaria_C2_Quota_Preset_Enc			:LREAL;
	Rotazione_C1_Quota_Preset_Enc			:LREAL;
	Rulliera_R1_Quota_Preset_Enc			:LREAL;
	Rulliera_R3_Quota_Preset_Enc			:LREAL;
	Rulliera_R2_Quota_Preset_Enc			:LREAL;
	Rotazione_C3_Quota_Preset_Enc			:LREAL;
	Rotazione_C5_Quota_Preset_Enc			:LREAL;
	Rotazione_C6_Quota_Preset_Enc			:LREAL;
	
	C1_Gap_Pezzi							:REAL;
	C2_Gap_Pezzi							:REAL;
	C3_Gap_Pezzi							:REAL;
	C5_Gap_Pezzi							:REAL;
	C6_Gap_Pezzi							:REAL;
	C1_Spazio_Libero_Start_Scarico			:REAL;
	
	R1_Lunghezza_Rulliera					:REAL;
	R2_Step_Value							:REAL;
	R3_Lunghezza_Rulliera					:REAL;
	C3_Lunghezza_Catenaria					:REAL;
	C4_Lunghezza_Catenaria					:REAL;
	C5_Lunghezza_Catenaria					:REAL;
		
	C1_Ribalta_Step_Fw						:REAL;
	C1_Ribalta_Step_Bk						:REAL;
	
	R2_Step_800_1000mm						:REAL;
	R2_Step_1001_2000mm						:REAL;
	R2_Step_2001_3500mm						:REAL;
	R2_Step_3500_9800mm						:REAL;
	R2_Step_9800mm							:REAL;
		
	
	Buffer_C1						: ARRAY [0..20] OF dut_Dati_Pezzo;
	Buffer_C2						: ARRAY [0..20] OF dut_Dati_Pezzo;
	Buffer_R1						: ARRAY [0..20] OF dut_Dati_Pezzo;
	Buffer_R2						: ARRAY [0..20] OF dut_Dati_Pezzo;
	Buffer_R3						: ARRAY [0..20] OF dut_Dati_Pezzo;
	Buffer_C3						: ARRAY [0..20] OF dut_Dati_Pezzo;
	Buffer_C4						: ARRAY [0..20] OF dut_Dati_Pezzo;
	Buffer_C5						: ARRAY [0..20] OF dut_Dati_Pezzo;
	Buffer_C6						: ARRAY [0..20] OF dut_Dati_Pezzo;
	
	Tempo_Svuotamento_Hdd			:TIME;
	
	R1_Set_Rotazione			:INT;   //99=no rotazione - 1=rot. avanti - 2=rot. indietro - 3=doppia rotazione
	R1_Set_Larghezza			:REAL;
	R1_Set_Altezza				:REAL;
	R1_Set_Lunghezza			:REAL;
	R1_Set_Lato_Scarico			:INT;	//1=destra - 2=sinistra
	R1_Set_Nr_Ricetta			:INT;
	
END_VAR

(*---------------------------------------------------------------------------   ------------------------------------------------------*)	
(*---------------------------------------------------------------------------   ------------------------------------------------------*)
(*---------------------------------------------------------------------------   ------------------------------------------------------*)

// ---- POUs/EVACUAZIONE_SCARTI/MAIN.TcPOU
PROGRAM MAIN
VAR
END_VAR


EVACUAZIONE_SCARTI();


//RULLI_CENTRO_TAGLI();

//GESTIONE_ASSI();

END_PROGRAM

// ---- POUs/EVACUAZIONE_SCARTI/EVACUAZIONE_SCARTI.TcPOU
PROGRAM EVACUAZIONE_SCARTI
VAR

	bINIT					:BOOL;
	
	//act Area MACINATORE
	rtAuto_ON				:R_TRIG;
	ftAuto_ON				:F_TRIG;
	tmrT3_ON				:TON;	
	tmrT3_OFF				:TON;		
	tmrT1T2_ON				:TON;	
	tmrT1T2_OFF				:TON;
	ft_AbilitaT1T2			:F_TRIG;
	ft_AbilitaT3			:F_TRIG;
	ft_AbilitaT4			:F_TRIG;
	
	Area_HS_On				:BOOL;
	rt_Area_M_Riarmo		:R_TRIG;
	rt_Area_M_Disarmo		:R_TRIG;
	tmr_SvuotaT1			:TON;		
	tmr_SvuotaT2			:TON;	
	tmr_SvuotaT3			:TON;	
	tmr_MacinatoreON		:TON;
	tmr_MacinatoreOFF		:TON;
	rt_MacinatoreON			:R_TRIG;
	rt_MacinatoreOFF		:R_TRIG;
	rt_MPO1_btn_M_MacOn		:R_TRIG;
	rt_btn_Fsx_T3StartMan	:R_TRIG;
	rt_btn_Fdx_T4StartMan	:R_TRIG;
	tmr_T3T5T6DelayStart	:TON;
	rt_T3S1full				:R_TRIG;
	tmr_T3S1vuoto			:TON;
	tmr_T3S1pieno			:TON;
	bT3S1full				:BOOL;
	rt_T3S2full				:R_TRIG;
	tmr_T3S2vuoto			:TON;
	bT3S2full				:BOOL;
	ft_T3S2full				:F_TRIG;
	countT3avanzamento		:INT;
	
	//act AREA SILOS
	rt_Area_S_Riarmo		:R_TRIG;
	rt_Area_S_Disarmo		:R_TRIG;
	
	//act_ALARM
	rtAlarmReset			:R_TRIG;	
	AlarmActive				:BOOL;
	AlarmReset				:BOOL;
	AlarmMask				:DWORD;
	T5_Bloccato				:ES_ALARM;	
	T6_Bloccato				:ES_ALARM;
	tmr_T4ON				:TON;
	
	tmrT3_Lavoro			:TON;	
	tmrT3_Pausa				:TON;
	tmrT5T6_RitStop			:TOF;	
	tmrS1_T_Rit_Empty		:TOF;
	tmrT1S01_Full			:TON;
	tmr_T_Rit_Stop_T4T5T6	:TOF;
	
	Forza_TT1S01_Full		:BOOL;
	
	appT1S01_Full			: BOOL;
	
	En_T_RitStopT5T6		:BOOL;
	
	//SENSORI	
	S1						:ES_S1;
	S2						:ES_S2;
	T1						:ES_T1;
	T3						:ES_T3;
	T5						:ES_T5;
	T6						:ES_T6;
                        	
	T1SO1tmravg				:TON;
	T1SO1arravg				:ARRAY[0..99]OF INT;
	T1SO1maxCnt				:INT;
	T1SO1sumavg				:REAL;
	T1SO1avg				:REAL;
	T1SO1cnt				:INT;
	T1SO1cnt2				:INT;	
	T1SO1cnt3				:INT;
	                    	
	S1SO2tmravg				:TON;
	S1SO2arravg				:ARRAY[0..99]OF INT;
	S1SO2maxCnt				:INT;
	S1SO2sumavg				:REAL;
	S1SO2avg				:REAL;
	S1SO2cnt				:INT;
	S1SO2cnt2				:INT;	
	S1SO2cnt3				:INT;		
                        	
	T3S1tmravg				:TON;
	T3S1arravg				:ARRAY[0..99]OF INT;
	T3S1maxCnt				:INT;
	T3S1sumavg				:REAL;
	T3S1avg					:REAL;
	T3S1cnt					:INT;
	T3S1cnt2				:INT;	
	T3S1cnt3				:INT;
	                    	
	T3S2tmravg				:TON;
	T3S2arravg				:ARRAY[0..99]OF INT;
	T3S2maxCnt				:INT;
	T3S2sumavg				:REAL;
	T3S2avg					:REAL;
	T3S2cnt					:INT;
	T3S2cnt2				:INT;	
	T3S2cnt3				:INT;
	                    	
	//SEMAFORI          	
	fbS1_Se1				:FB_Semaforo;
		
	//gestione filtro temporale sensore 
	SO2_full_curr			:BOOL;
	tmrValidaSoglia_S02		:TON;

	
	//gestione macinatore
	TON_Macinatore_On			:TON;
	TON_Vibro_Macinatore_On		:TON;
	TON_Ciclo_Macinatore		:TON;
	TP_Start_Macinatore			:TP;
	TP_Stop_Macinatore			:TP;

	TS							:BOOL;
	M_Ciclo_Svuotamento_Hdd_RUN	:BOOL;
	M_Auto_Start_Macinatore		:BOOL;
	M_Auto_Start_Vibro_Macinatore		:BOOL;
	M_Auto_Start_Vibro_Hdd		:BOOL;
	M_Start_Req_Stop_Macinatore	:BOOL;	
	M_Stop_Req_Stop_Macinatore	:BOOL;
	
	M_Man_Start_Vibro_Hdd		:BOOL;
	
	
	
	
	//TwinsAFE
	tmrErrAck				:TON;	
	
END_VAR
VAR // added by the converter: edge detectors and wires of the graphical bodies
    _rt1, _rt2 : R_TRIG;
    _w1, _w2, _w3 : BOOL;
    _ft1 : F_TRIG;
END_VAR


act_INIT();

act_ALARM();

act_INPUT();

act_Sensori();

act_AreaSilos();

act_Macinatore();

//act_AreaMac_AUTO();
//act_AreaMac_MAN();

act_Semafori();

act_OUTPUT();

act_HMI();

ACTION act_ALARM:

//TwinSAFE
TS_ErrAck := C1P1_Rst_Eme OR R1P1_Rst_Eme;


tmrErrAck(IN:=TS_ErrAck,PT:=T#1S);
IF tmrErrAck.Q THEN
	TS_ErrAck:=FALSE;
END_IF




//ALLARMI DA SENSORI
rtAlarmReset(CLK:=bAlarmReset);
IF rtAlarmReset.Q THEN
	bAlarmReset:=FALSE;
	T5.Alarm.Active:=FALSE;	
	T6.Alarm.Active:=FALSE;	
	bAllarmeT5:=FALSE;
	bAllarmeT6:=FALSE;
END_IF

IF NOT AlarmActive THEN

	//Allarme T5 Bloccato - 5s
	IF HQ1_T5_KA5 THEN
		T5.Alarm.tmr(IN:=TRUE,PT:=INT_TO_TIME(T5.Alarm.pt*1000));
		IF T5.Alarm.tmr.ET < T5.Alarm.tmr.PT THEN
			T5.S1_rt(CLK:=T5_S1);
			IF T5.S1_rt.Q THEN
				T5.S1_letto:=TRUE;		
			END_IF
		END_IF
	
		IF T5.Alarm.tmr.Q THEN
			IF NOT T5.S1_letto AND HQ1_T5_KA5 THEN
				T5.Alarm.Active:=TRUE AND bAllarmeT5enable;	
			ELSE	
				T5.Alarm.Active:=FALSE;	
			END_IF
			T5.S1_letto:=FALSE;
			T5.Alarm.tmr(IN:=FALSE);
		END_IF
	END_IF

	
	
		
	//Allarme T6 Bloccato - 5s
	IF HQ1_T6_KA6 THEN
		T6.Alarm.tmr(IN:=TRUE,PT:=INT_TO_TIME(T6.Alarm.pt*1000));
		IF T6.Alarm.tmr.ET < T6.Alarm.tmr.PT THEN
			T6.S1_rt(CLK:=T6_S1);
			IF T6.S1_rt.Q THEN
				T6.S1_letto:=TRUE;		
			END_IF
		END_IF
	
		IF T6.Alarm.tmr.Q THEN
			IF NOT T6.S1_letto AND HQ1_T6_KA6 THEN
				T6.Alarm.Active:=TRUE AND bAllarmeT6enable;	
			ELSE	
				T6.Alarm.Active:=FALSE;	
			END_IF
			T6.S1_letto:=FALSE;
			T6.Alarm.tmr(IN:=FALSE);
		END_IF	
	END_IF
	

	
	
	//Allarme S2 Silos Pieno
	IF S2.S1_full (*AND glo_ES_BtnHMI.S2_Alarm_Enable*) THEN
		S2.Alarm.Active := TRUE AND bAllarmeS2S1enable;
	END_IF
	
	
	
	
	//Allarme T3 Bloccato - 30s
	IF T1.SO1_full AND T3.S1_full THEN
		T3.Alarm.tmr(IN:=TRUE,PT:=INT_TO_TIME(T3.Alarm.pt*1000));
		IF T3.Alarm.tmr.Q THEN
			T3.Alarm.tmr(IN:=FALSE);
			T3.Alarm.Active := TRUE;	
		END_IF
	ELSE
		T3.Alarm.Active := FALSE;
	END_IF	

	
	
	
	//Allarme S1 Silos1 Pieno
	IF (*S1_S2_full AND*) S1_S2 THEN
		S1.Alarm.Active:=TRUE;
	END_IF
	
END_IF
END_ACTION

ACTION act_AreaMac_AUTO:

//#######################################################
//###################    AREA M ON    ###################
//#######################################################

IF M_PO1.key THEN
	rt_Area_M_Riarmo(CLK:= M_PO1.btn_R_Riarmo OR bSIMULA_btnR);
	IF rt_Area_M_Riarmo.Q THEN
		bSIMULA_btnR:=FALSE;
		AreaM_ON:= TRUE;
	END_IF
END_IF
rt_Area_M_Disarmo(CLK:= M_PO1.btn_0_AreaMoff OR bSIMULA_btn0);
IF NOT M_PO1.key OR rt_Area_M_Disarmo.Q OR NOT TS_AreaM_ON OR NOT TS_AreaS_ON (*OR NOT TS_AreaM_OFF*) THEN
	bSIMULA_btn0:=FALSE;	
	AreaM_ON:=FALSE;
	fun_AreaM_SPEGNITUTTO();	
END_IF

//#######################################################
//##################     AUTOMATICO   ###################
//#######################################################

rtAuto_ON(CLK:=HQ1_Auto_ON OR bSIMULAAuto_ON);
IF rtAuto_ON.Q THEN
	bIsAuto:=TRUE;
END_IF
ftAuto_ON(CLK:=HQ1_Auto_ON OR bSIMULAAuto_ON);
IF ftAuto_ON.Q THEN
	bIsAuto:=FALSE;	
	bSIMULA_btn0:=TRUE;	
	bSIMULA_btn0silos:=TRUE;	
	fun_AreaM_SPEGNITUTTO();	
END_IF

IF bIsAuto THEN
	

	//#######################################################
	//####################     T1 - T2    ###################
	//#######################################################
	
	(*
	- sensore sotto hundegger dà che T1 è pieno
	- area attiva
	- sensore all'inizio del T3 dà che è vuoto/libero
	- T3 non è bloccato: sensori del T1 e T3 contemporaneamente non pieni
	*)
	
	IF bAbilitaT1T2 THEN
		
		CASE stepT1T2 OF
			
			0:
				descT1T2:='T1-T2 spenti. In attesa di T1SO1 pieno';
				IF T1.SO1_full THEN
					stepT1T2:=5;
				END_IF
			
			5:
				IF NOT T3.S1_full (*AND NOT T3.Alarm.Active*) THEN 
					descT1T2:='Avvio T1-T2';
					bT1_ON:=TRUE;
					bT2_ON:=TRUE;
					tmrT1T2_ON(IN:=FALSE);
					stepT1T2:=10;
				ELSIF T3.S1_full (*OR T3.Alarm.Active*) THEN
					stepT1T2:=100;
				END_IF
			
			10:
				descT1T2:='T1-T2 accesi per 2s';
				tmrT1T2_ON(IN:=TRUE,PT:=T#2S);
				IF tmrT1T2_ON.Q THEN
					tmrT1T2_OFF(IN:=FALSE);
					stepT1T2:=15;					
				END_IF
			
			15:
				descT1T2:='T1-T2 accesi finchè T3S1 pieno';		
				IF NOT T1.SO1_full THEN
					tmrT1T2_ON(IN:=FALSE);					
					bT1_ON:=FALSE;
					stepT1T2:=16;
				END_IF		
				tmr_T3S1pieno(in:=T3.S1_full,PT:=T#2S);
				IF tmr_T3S1pieno.Q THEN
					bT1_ON:=FALSE;
					bT2_ON:=FALSE;
					stepT1T2:=20;				
				END_IF
	
			16:
				descT1T2:='T1spento, T2 acceso per 15s o finchè T3S1 pieno';	
				tmrT1T2_ON(IN:=TRUE,PT:=T#15S);	
				IF tmrT1T2_ON.Q OR T3.S1_full THEN
					bT2_ON:=FALSE;
					stepT1T2:=20;
				END_IF	
		
			20:
				descT1T2:='T1-T2 spenti, pausa 30s';
				tmrT1T2_OFF(IN:=TRUE,PT:=T#30S);
				IF tmrT1T2_OFF.Q THEN
					stepT1T2:=100;						
				END_IF
			
			100:
				tmrT1T2_OFF(IN:=FALSE);
				tmrT1T2_ON(IN:=FALSE);
				bT1_ON:=FALSE;
				bT2_ON:=FALSE;
				stepT1T2:=0;
					
		END_CASE
			
	END_IF
	ft_AbilitaT1T2(CLK:=bAbilitaT1T2);
	IF ft_AbilitaT1T2.Q THEN
		descT1T2:='T1-T2 disabilitati';
		HQ1_T1_KA1:=FALSE;
		HQ1_T2_KA2:=FALSE;
		bT1_ON:=FALSE;
		bT2_ON:=FALSE;
		stepT1T2:=100;			
	END_IF
	
	
	
	//#######################################################
	//##############    M - T3 - T5 - T6    #################
	//#######################################################
	
	(*
	- area attiva
	- bottone Macinatore da pulsantiera (vedi sotto fuori dall'automatico)
	- sensore all'inizio del T3 dà che è pieno
	- Silos2 non deve essere pieno
	- T5 non bloccato controllo paletta
	- T6 non bloccato controllo paletta
	*)
	IF NOT bAbilitaT3 THEN
		
		countT3avanzamento:=0;
		
	END_IF
	
	IF bAbilitaT3 THEN
	
		//azzeramento step automatici se il macinatore è stato avviato in locale
	//	IF NOT M_Start_Macinatore_Loc THEN
		//	stepT3 :=0;
	//	END_IF;
		CASE stepT3 OF
			
			0:
				descT3:='T3 fermo. In attesa di T3S1 pieno';
				IF NOT bT4_ON THEN// AND NOT M_Start_Macinatore_Loc THEN
					tmrT3_OFF(IN:=FALSE);
					tmrT3_ON(IN:=FALSE);
					IF T3.S1_full THEN	
						//PIENO INGRESSO, USCITA SCARICA -> ACCENDO T3						
						tT3ON_auto:=15;
						IF countT3avanzamento >=5 THEN
							descT3:='Macinatore acceso, attendo 20s per avvio T3';
							bM_ON:=TRUE;
							stepT3:=10;	
						ELSE
							descT3:='T3 acceso per 30s';
							bT3_ON:=TRUE;
							stepT3:=5;	
						END_IF	
					END_IF
				END_IF
		
			5:
				descT3:='T3 acceso per 30s';
				bT3_ON:=TRUE;
				tmrT3_ON(IN:=TRUE,PT:=INT_TO_TIME(tT3ON_auto*1000));
				IF tmrT3_ON.Q OR T3.S2_full THEN
					bT3_ON:=FALSE;	
					tmrT3_OFF(IN:=FALSE);
					countT3avanzamento:=countT3avanzamento+1;
					stepT3:=20;
				END_IF	
			
			10:
				descT3:='Macinatore acceso, attendo 20s per avvio T3';
				tmrT3_OFF(IN:=TRUE,PT:=T#20S);
				IF tmrT3_OFF.Q THEN
					bT3_ON:=TRUE;
					T3_ModoPausaLavoro:=TRUE;
					bT3EnT1PausaLavoro:=TRUE;  (*abilito un timer per far lavorare T3 pausa-lavoro per non intasare T5*)
					bT3EnT2PausaLavoro:=FALSE;
					T3_Lavoro:=TRUE;
					stepT3:=15;
				END_IF
		
			15:
				descT3:='T3 e Macinatore accesi per 5min';
				tmrT3_ON(IN:=TRUE,PT:=T#8M);
				IF tmrT3_ON.Q THEN
					tmrT3_OFF(IN:=FALSE);
					bM_ON:=FALSE;
					bT3_ON:=FALSE;
					T3_ModoPausaLavoro:=FALSE;
					bT3EnT1PausaLavoro:=FALSE;
					bT3EnT2PausaLavoro:=FALSE;
					T3_Lavoro:=FALSE;
					stepT3:=20;
					countT3avanzamento:=0;
				END_IF
				
			20:
				descT3:='Tutto spento, pausa di 30s';
				tmrT3_OFF(IN:=TRUE,PT:=T#30S);
				IF tmrT3_OFF.Q THEN
					tmrT3_OFF(IN:=FALSE);
					stepT3:=0;
				END_IF
			
			100:
				tmrT3_OFF(IN:=FALSE);
				tmrT3_ON(IN:=FALSE);
				bM_ON:=FALSE;
				stepT3:=0;
		
		END_CASE
	
	END_IF
	ft_AbilitaT3(CLK:=bAbilitaT3);
	IF ft_AbilitaT3.Q THEN
		descT3:='T3 disabilitato';
		HQ1_T3_KA3:=FALSE;	
		bMacinatoreStart:=FALSE;
		bMacinatoreStop:=TRUE;
		stepT3:=100;		
	END_IF
	
	
	
	//#######################################################
	//#################     T4 - T5 - T6    #################
	//#######################################################
	
	(*
	- T5 non bloccato controllo paletta
	- T6 non bloccato controllo paletta
	- Silos2 non deve essere pieno
	- Consenso da logica Aspirazione
	*)
	
	IF bAbilitaT4 THEN
		
		CASE stepT4 OF
			
		0:
			descT4:='T4 fermo. In attesa di LogicaAspirazioneON';
			IF (NOT bT3_ON AND bMacinatoreStop) AND LogicaAspirazioneON THEN
				bT4_ON:=TRUE;
				stepT4:=10;
			END_IF
		
		10:
			descT4:='T4 acceso per 30s';
			tmr_T4ON(IN:=TRUE,PT:=T#30S);	
			IF tmr_T4ON.Q THEN
				tmr_T4ON(IN:=FALSE);
				IF NOT LogicaAspirazioneON THEN
					stepT4:=100;			
				END_IF				
			END_IF
			
		100:
			tmr_T4ON(IN:=FALSE);
			bT4_ON:=FALSE;
			stepT4:=0;
					
		END_CASE

	END_IF
	ft_AbilitaT4(CLK:=bAbilitaT4);
	IF ft_AbilitaT4.Q THEN
		descT4:='T4 disabilitato';
		HQ1_T4_KA4:=FALSE;
		bT4_ON:=FALSE;
		stepT4:=100;			
	END_IF
	
END_IF



//####################################################################
//####     GESTIONE TIMER PAUSA LAVORO IN CICLO AUTOMATICO T3 #######
//###################################################################

tmrT3_Lavoro(IN:=bT3EnT1PausaLavoro,PT:=T#20S);
tmrT3_Pausa(IN:=bT3EnT2PausaLavoro,PT:=T#30S);

IF tmrT3_Lavoro.Q THEN
	bT3EnT1PausaLavoro := FALSE;	
	bT3EnT2PausaLavoro := TRUE;
	T3_Lavoro := FALSE;	
END_IF

IF tmrT3_Pausa.Q THEN
	bT3EnT1PausaLavoro := TRUE;	
	bT3EnT2PausaLavoro := FALSE;
	T3_Lavoro := TRUE;
END_IF

//##################################################################
//####     		 GESTIONE TIMER RITARDO STOP T5-T6	 		 #######
//##################################################################
En_T_RitStopT5T6 := bM_ON AND AreaM_ON;
tmrT5T6_RitStop(IN:=En_T_RitStopT5T6,PT:=T#30S);

//#######################################################
//####     USCITE INDIPENDENDI DA MODO AUTO/MAN   #######
//#######################################################

HQ1_T1_KA1:= bT1_ON AND AreaM_ON;
HQ1_T2_KA2:= bT2_ON AND AreaM_ON;

M_Cmd_T3 := bT3_ON AND (T3_Lavoro OR NOT T3_ModoPausaLavoro);

HQ1_T3_KA3:= M_Cmd_T3 AND NOT SensInMac AND AreaM_ON AND NOT (T5.Alarm.Active OR T6.Alarm.Active OR S2.Alarm.Active);		
HQ1_T4_KA4:= bT4_ON AND AreaM_ON AND LogicaAspirazioneON AND NOT (T5.Alarm.Active OR T6.Alarm.Active OR S2.Alarm.Active);
HQ1_T5_KA5:= (bM_ON OR bT4_ON OR tmrT5T6_RitStop.Q) AND AreaM_ON AND NOT (T5.Alarm.Active OR T6.Alarm.Active OR S2.Alarm.Active);
HQ1_T6_KA6:= (bM_ON OR bT4_ON OR tmrT5T6_RitStop.Q) AND AreaM_ON AND NOT T6.Alarm.Active AND NOT S2.Alarm.Active;
		

bMacinatoreStart:= bM_ON AND AreaM_ON AND NOT (T5.Alarm.Active AND T6.Alarm.Active AND S2.Alarm.Active) and HQ1_T5_KA5;
bMacinatoreStop:= NOT bM_ON OR T5.Alarm.Active OR T6.Alarm.Active OR NOT HQ1_T5_KA5 OR NOT HQ1_T5_KA5;	

//#######################################################
//#############     START-STOP MACINATORE   #############
//#######################################################

//AVVIO MACINATORE RICHIEDE CHE DOPO 1s USCITA VENGA ABBASSATA
rt_MacinatoreON(CLK:=bMacinatoreStart);	
IF rt_MacinatoreON.Q THEN
	HQ1_M_ON:=TRUE;
	HQ1_M_OFF:=FALSE;

END_IF
tmr_MacinatoreON(IN:=HQ1_M_ON,PT:=T#1S);	
IF tmr_MacinatoreON.Q THEN
	tmr_MacinatoreON(IN:=FALSE);
	HQ1_M_ON:=FALSE;
END_IF
//SPEGNIMENTO MACINATORE RICHIEDE CHE DOPO 1s USCITA VENGA ABBASSATA
rt_MacinatoreOFF(CLK:=bMacinatoreStop);	
IF rt_MacinatoreOFF.Q THEN
	HQ1_M_ON:=FALSE;
	HQ1_M_OFF:=TRUE;

END_IF
tmr_MacinatoreOFF(IN:=HQ1_M_OFF,PT:=T#1S);	
IF tmr_MacinatoreOFF.Q THEN
	tmr_MacinatoreOFF(IN:=FALSE);
	HQ1_M_OFF:=FALSE;
END_IF
	
		
	
	

//#######################################################
//##################     PULSANTIERA   ##################
//#######################################################

IF AreaM_ON AND bAbilitaPulsatiera THEN
	
	//M	
	rt_MPO1_btn_M_MacOn(CLK:=(M_PO1.btn_M_MacOn OR bSIMULA_btnM));
	IF rt_MPO1_btn_M_MacOn.Q AND bMacinatoreStop THEN
		bSIMULA_btnM:=FALSE;
		//M SPENTO -> LO ACCENDO
		bM_ON:=TRUE;
		IF NOT SensInMac AND NOT HQ1_T4_KA4 THEN
			bT3T5T6DelayStart:= TRUE;
		END_IF		
	ELSIF rt_MPO1_btn_M_MacOn.Q AND bMacinatoreStart THEN
		//M ACCESO -> LO SPENGO
		bSIMULA_btnM:=FALSE;
		bM_ON:=FALSE;	
		bT3T5T6DelayStart:=FALSE;
		IF (*NOT M_PO1.btn_Fsx_T3StartMan AND*) NOT glo_ES_ActVal.PuliziaT1t2_ON THEN
			bT3_ON:=FALSE;
			M_Start_Macinatore_Loc := FALSE;
		END_IF
	END_IF
	
	IF (T5.Alarm.Active OR T6.Alarm.Active OR S2.Alarm.Active) THEN
		bM_ON:=FALSE;
	END_IF
		
	//AVVIO RITARDATO DEL T3,T5,T6 DOPO 15s DALL'AVVIO M	
	tmr_T3T5T6DelayStart(IN:=bT3T5T6DelayStart, PT:=T#35S);
	IF tmr_T3T5T6DelayStart.Q THEN
		bT3T5T6DelayStart:=FALSE;
		bT3_ON:=TRUE;
		M_Start_Macinatore_Loc := TRUE;
	END_IF
	
	//T3
	rt_btn_Fsx_T3StartMan(CLK:=M_PO1.btn_Fsx_T3StartMan OR bSIMULA_btnT3);		//FRECCIA A SINISTRA SU BOTTONE DI SINISTRA
	IF rt_btn_Fsx_T3StartMan.Q THEN
		IF NOT SensInMac AND NOT HQ1_T3_KA3 THEN				//SE SENSORE SU MAC è ON, ALLORA NN ACCENDO T3 XKE LO INTASO
			bSIMULA_btnT3:=FALSE;
			bT3_ON:= TRUE;
		ELSIF NOT glo_ES_ActVal.PuliziaT1t2_ON AND HQ1_T3_KA3 THEN
			bSIMULA_btnT3:=FALSE;
			bT3_ON:=FALSE;
		END_IF			
	END_IF
	
	IF NOT bM_ON THEN 
		bT3_ON:=FALSE;
	END_IF
	
	//T4
	rt_btn_Fdx_T4StartMan(CLK:=M_PO1.btn_Fsx_T4StartMan);
	IF rt_btn_Fdx_T4StartMan.Q THEN		//FRECCIA A SINISTRA SU BOTTONE DI DESTRA
		IF NOT HQ1_T4_KA4 THEN	
			bT4_ON:= TRUE;
		ELSE
			bT4_ON:=FALSE;
		END_IF
	END_IF
		
	//T7
	IF M_PO1.btn_Fup_T7Avanti THEN			//FRECCIA IN SU
		HQ1_T7_A_KA8:= TRUE;
		HQ1_T7_I_KA9:= FALSE;
	ELSIF M_PO1.btn_Fdw_T7Indietro THEN		//FRECCIA IN GIU'
		HQ1_T7_I_KA9:= TRUE;
		HQ1_T7_A_KA8:=FALSE;
	ELSE
		HQ1_T7_A_KA8:=FALSE;
		HQ1_T7_I_KA9:= FALSE;
	END_IF
	
END_IF
END_ACTION

ACTION act_AreaMac_MAN:

//#######################################################
//####################     MANUALE   ####################
//#######################################################


IF NOT bIsAuto THEN
		
	//#######################################################
	//###############     PULIZIA T1-T2-T3   ################
	//#######################################################

	IF 	bMAN_SvuotaT1T2T3 THEN
		bMAN_SvuotaT1T2T3:=FALSE;
		glo_ES_ActVal.PuliziaT1T2_ON:=TRUE;
		bT1_ON:= TRUE;
		bT2_ON:= TRUE;
		bM_ON:= TRUE;
		bT3T5T6DelayStart:=TRUE;
	END_IF
	IF glo_ES_ActVal.PuliziaT1T2_ON THEN
		tmr_SvuotaT1(IN:= bT1_ON,PT:=DINT_TO_TIME(glo_ES_Config.T1_Time*1000));
		tmr_SvuotaT2(IN:= bT2_ON,PT:=DINT_TO_TIME(glo_ES_Config.T2_Time*1000));
		tmr_SvuotaT3(IN:= bM_ON,PT:=DINT_TO_TIME(glo_ES_Config.T3_Time*1000));
	END_IF

	//STOP T1
	IF tmr_SvuotaT1.Q THEN
		tmr_SvuotaT1(IN:=FALSE);
		bT1_ON:= FALSE;
	END_IF
		
	//STOP T2
	IF tmr_SvuotaT2.Q THEN
		tmr_SvuotaT2(IN:=FALSE);
		bT2_ON:= FALSE;
	END_IF
	
	//STOP T3	
	IF tmr_SvuotaT3.Q THEN
		tmr_SvuotaT3(IN:=FALSE);
		bM_ON:= FALSE;
		bT3T5T6DelayStart:=FALSE;
		glo_ES_ActVal.PuliziaT1t2_ON:=FALSE;
	END_IF

	
	//#######################################################
	//#################     PULIZIA S1-T4   #################
	//#######################################################
	
	IF bMAN_SvuotaS1T4 THEN
		bMAN_SvuotaS1T4:=FALSE;
		
	END_IF
	
	
END_IF
END_ACTION

ACTION act_AreaSilos:

//#######################################################
//###################    AREA S ON    ###################
//#######################################################

IF S1_PO1.key THEN
	rt_Area_S_Riarmo(CLK:= S1_PO1.btn_R_Riarmo OR bSIMULA_btnRsilos);
	IF rt_Area_S_Riarmo.Q THEN
		bSIMULA_btnRsilos:=FALSE;
		AreaS_ON:= TRUE;
	END_IF
END_IF
rt_Area_S_Disarmo(CLK:= S1_PO1.btn_0_AreaMoff OR bSIMULA_btn0silos);
IF NOT S1_PO1.key OR rt_Area_S_Disarmo.Q OR NOT TS_AreaM_ON OR NOT TS_AreaS_ON (*OR TS_AreaS_OFF*) THEN
	bSIMULA_btn0silos:=FALSE;	
	AreaS_ON:=FALSE;
END_IF

	//led pulsante area macinatore ON
	S1_PO1.led_0_AreaMoff := AreaS_ON;

	//led pulsante riarmo area macinatore
	S1_PO1.led_R_Riarmo := TS_AreaS_ON;
	
	//riarmo emergenze
//	TS_S1PO1_btn_R := S1_PO1.key AND S1_PO1.btn_R_Riarmo;
	TS_S1PO1_btn_R := S1_PO1.key AND(C1P1_Rst_Eme OR R1P1_Rst_Eme);
	
	
//#######################################################
//#############    LOGICA M-ASPIRAZIONE   ###############
//#######################################################

IF AreaS_ON AND bAbilitaPulsatieraS1PO1 THEN
	
	//VALVOLA STELLARE S1_SO2	
	IF (S1.SO2_full) AND NOT bT3_ON AND bMacinatoreStop AND NOT bSIMULA_BrichettatriceON AND bAbilitaT4 THEN
		HQ1_S1_ValvolaStellare:=TRUE;
	ELSE
		HQ1_S1_ValvolaStellare:=FALSE;
	END_IF
	
//	HQ1_S1_ValvolaStellare:=FALSE;
	
	//BRICCHETTATRICE
	IF (*HQ1_ScorniciatriceON AND NOT HQ1_S1_ValvolaStellare AND*) bSIMULA_BrichettatriceON THEN
		HQ1_BrichettatriceON:=TRUE;
	ELSE
		HQ1_BrichettatriceON:=FALSE;
	END_IF
	
	//RACLA
	IF HQ1_BrichettatriceON OR HQ1_S1_ValvolaStellare THEN
		HQ1_RaclaON:=TRUE;
	ELSE
		HQ1_RaclaON:=FALSE;
	END_IF 
	
	//CONSENSO A T4 T5 T6
tmr_T_Rit_Stop_T4T5T6(IN:=HQ1_S1_ValvolaStellare,PT:=T#1M);
	
IF tmr_T_Rit_Stop_T4T5T6.Q THEN
		LogicaAspirazioneON:=TRUE;
	ELSE
		LogicaAspirazioneON:=FALSE;		
	END_IF
	
END_IF
END_ACTION

ACTION act_HMI:


bAllarmeT3	:= T3.Alarm.Active;			
bAllarmeT5	:= T5.Alarm.Active;			
bAllarmeT6	:= T6.Alarm.Active;
bAllarmeS2S1:= S2.Alarm.Active;

bT1SO1pieno	:= T1.SO1_full;
bT3S1pieno	:= T3.S1_full;
bT3S2pieno	:= T3.S2_full;
bS1SO2pieno	:= S1.SO2_full;
bS2S1pieno	:= S2.S1_full;

glo_ES_ActVal.T3_S1:= T3.S1_actVal;
glo_ES_ActVal.T3_S2:= T3.S2_actVal;
glo_ES_ActVal.S2_S1:= S2.S1_actVal;
glo_ES_ActVal_T1_SO1:= T1_SO1;

altMatT3S1:=T3.S1_fb.distanzaAVuoto - T3.S1_actVal;
IF altMatT3S1 <0 THEN
	altMatT3S1:=0;
END_IF
altMatT3S2:=T3.S2_fb.distanzaAVuoto - T3.S2_actVal;
IF altMatT3S2 <0 THEN
	altMatT3S2:=0;
END_IF 
distMatT1SO1:= T1.SO1_fb.distanzaAVuoto - T1.SO1_actVal;
IF distMatT1SO1 <0 THEN
	distMatT1SO1:=0;
END_IF 

IF sogliaT3S1 = 0 THEN
	sogliaT3S1:=100;
END_IF
IF sogliaT3S2 = 0 THEN
	sogliaT3S2:=40;
END_IF
//IF sogliaS1SO2 = 0 THEN
//	sogliaS1SO2:=1000;
//END_IF
IF solgiaT1SO1 = 0 THEN
	solgiaT1SO1:=5000;
END_IF
END_ACTION

ACTION act_INIT:

IF NOT bINIT THEN
	
	bINIT:=TRUE;

	bMacinatoreStop:=TRUE;

	//Avvia TwinSAFE Gruppo EVACUAZIONE SCARTI
	TS_Run_GrpES:=TRUE;

END_IF
END_ACTION

ACTION act_INPUT:

//TERM7 EL1008 H-Q1
SensInMac				:= glo_dig_in_HQ1[1];		//DIGIN CH1			Sensore ingresso macinatore
R5_S2					:= glo_dig_in_HQ1[2];		//DIGIN CH2			Val1 aperta
T5_S3					:= glo_dig_in_HQ1[3];		//DIGIN CH3			Val2 chiusa
S1_S3					:= glo_dig_in_HQ1[4];		//DIGIN CH4			Allarme silos1 pieno
T6_S1					:= glo_dig_in_HQ1[5];		//DIGIN CH5			Rotaz catena IFS289
HQ1_Auto_ON				:= glo_dig_in_HQ1[6];		//DIGIN CH6			Modo auto-man
HQ1_P1					:= glo_dig_in_HQ1[7];		//DIGIN CH7			Reset Allarme
HQ1_K1					:= glo_dig_in_HQ1[8];		//DIGIN CH8			---

//TERM8 EL1008 H-Q1
//HQ1_AspirazioneON		:= glo_dig_in_HQ1[10];		//DIGIN CH2			Motore aspirazione in silos S1
I_Fdbk_Km_Area_Nastri_Macinatore:= glo_dig_in_HQ1[9];		//DIGIN CH2			feedback contattore area macinatore
I_Fdbk_Km_Area_Macinatore:= glo_dig_in_HQ1[10];		//DIGIN CH2			feedback contattore area macinatore
I_Macinatore_Run		:= glo_dig_in_HQ1[12];		//DIGIN CH1			Scorniciatrice accesa

S1_S2					:= glo_dig_in_HQ1[12];		//DIGIN CH4			Sensore troppopieno in alto in silos S1
S1_S1					:= glo_dig_in_HQ1[13];		//DIGIN CH5			Sensore livello in basso in silos S1
HQ1_BricchettatriceON	:= glo_dig_in_HQ1[13];		//DIGIN CH6			Bricchettatrice accesa



//TERM11 EL3012 H-Q1
T3_S1					:= glo_analog_in_HQ1[1];	//ANALOGIN CH1		Pres materiale In T3
T3_S2					:= glo_analog_in_HQ1[2];	//ANALOGIN CH2		Pres materiale Out T3

//TERM12 EL3012 H-Q1
S1_SO2					:= glo_analog_in_HQ1[3];	//ANALOGIN CH1		Liv silos2 UMT 30-6000


(*****************************************************************)	
(*****************************************************************)	
(*****************************************************************)

//BOX16 EP6228-0022 M-CS1
T1_SO1					:= glo_analog_in_MCS1[1];	//IOLINK CH1	Già in mm. Pres mat T1, da inizio vibro fino sopra nastro  O1D120


(*****************************************************************)	
(*****************************************************************)	
(*****************************************************************)

//BOX17 EP6228-0022 T3-C01
S2_S1					:= glo_analog_in_T3C01[1];	//IOLINK CH2		LIV AVVIO VALV STELLARE UGT514

//S1_PO1											//IOLINK CH3		PULSANTIERA BNI005N
S1_PO1.key				:= glo_dig_in_T3C01[1];		//CHIAVE
S1_PO1.btn_0_AreaMoff	:= glo_dig_in_T3C01[2];		//BOTTONE '0'
S1_PO1.btn_R_Riarmo		:= glo_dig_in_T3C01[3];		//BOTTONE 'r'
I_Pls_Start_Vibro_Hdd	:= glo_dig_in_T3C01[7];

//M_PO1												//IOLINK CH4		PULSANTIERA BNI005M
M_PO1.key				:= glo_dig_in_T3C01[1];		//CHIAVE
M_PO1.btn_0_AreaMoff	:= glo_dig_in_T3C01[2];	//BOTTONE '0'
M_PO1.btn_R_Riarmo		:= glo_dig_in_T3C01[3];	//BOTTONE 'r'
M_PO1.btn_M_MacOn		:= glo_dig_in_T3C01[4];	//TASTO 'M'
M_PO1.btn_Fdw_T7Indietro:= glo_dig_in_T3C01[13];	//FRECCIA IN GIU'
M_PO1.btn_Fup_T7Avanti	:= glo_dig_in_T3C01[14];	//FRECCIA IN SU
M_PO1.btn_Fsx_T3StartMan:= glo_dig_in_T3C01[15];	//FRECCIA SX BTN SX
M_PO1.btn_Fsx_T4StartMan:= glo_dig_in_T3C01[16];	//FRECCIA SX BTN DX

T5_S1					:= glo_dig_in_T3C01[25];	//DIGIN  CH7		ROTAZ CATENA IFS289
T5_SO1					:= glo_analog_in_T3C01[2];	//IOLINK CH8		LIV SCARICO MAC UGT525

//
I_Barriera_Macinatore := glo_dig_in_T3C01[10];
END_ACTION

